C07285=1071.628,278.131,410.233,174.317,29.614,155.314
C07286=1071.623,277.882,410.263,174.314,29.610,155.313
C07287=1071.617,277.634,410.293,174.312,29.606,155.313
C07288=1071.611,277.386,410.322,174.309,29.602,155.312
C07289=1071.601,276.969,410.372,174.304,29.595,155.311
C07290=1071.591,276.552,410.422,174.300,29.588,155.310
C07291=1071.581,276.135,410.472,174.295,29.581,155.309
C07292=1071.570,275.717,410.522,174.291,29.575,155.307
C07293=1071.565,275.469,410.552,174.288,29.570,155.307
C07294=1071.558,275.221,410.581,174.285,29.567,155.306
C07295=1071.553,274.973,410.611,174.283,29.562,155.305
C07296=1071.547,274.725,410.640,174.280,29.558,155.305
C07297=1071.541,274.476,410.670,174.278,29.554,155.304
C07298=1071.535,274.228,410.699,174.275,29.550,155.303
C07299=1071.529,273.980,410.729,174.272,29.547,155.303
C07300=1071.523,273.732,410.758,174.270,29.542,155.302
C07301=1071.517,273.484,410.788,174.267,29.538,155.301
C07302=1071.512,273.236,410.817,174.264,29.534,155.301
C07303=1071.506,272.988,410.846,174.261,29.530,155.300
C07304=1071.500,272.740,410.875,174.259,29.526,155.299
C07305=1071.494,272.491,410.905,174.256,29.522,155.299
C07306=1071.488,272.243,410.934,174.254,29.518,155.298
C07307=1071.483,271.995,410.963,174.251,29.514,155.297
C07308=1071.476,271.747,410.992,174.249,29.510,155.297
C07309=1071.470,271.499,411.022,174.246,29.506,155.296
C07310=1071.465,271.250,411.051,174.244,29.502,155.295
C07311=1071.458,271.002,411.080,174.241,29.498,155.295
C07312=1071.452,270.754,411.109,174.239,29.494,155.294
C07313=1071.447,270.505,411.139,174.235,29.490,155.293
C07314=1071.440,270.257,411.168,174.233,29.486,155.293
C07315=1071.435,270.009,411.198,174.230,29.482,155.292
C07316=1071.429,269.761,411.227,174.228,29.478,155.291
C07317=1071.422,269.513,411.256,174.225,29.474,155.291
C07318=1071.417,269.264,411.285,174.223,29.470,155.290
C07319=1071.411,269.017,411.314,174.220,29.466,155.289
C07320=1071.405,268.769,411.343,174.218,29.462,155.289
C07321=1071.399,268.520,411.371,174.215,29.458,155.288
C07322=1071.393,268.271,411.401,174.213,29.455,155.287
C07323=1071.387,268.023,411.430,174.210,29.450,155.287
C07324=1071.381,267.775,411.459,174.208,29.446,155.286
C07325=1071.375,267.527,411.488,174.205,29.442,155.285
C07326=1071.369,267.278,411.516,174.202,29.438,155.285
C07327=1071.363,267.030,411.546,174.200,29.434,155.284
C07328=1071.358,266.782,411.575,174.197,29.431,155.283
C07329=1071.351,266.534,411.604,174.195,29.427,155.283
C07330=1071.345,266.286,411.632,174.191,29.422,155.282
C07331=1071.340,266.037,411.662,174.189,29.419,155.282
C07332=1071.334,265.789,411.691,174.186,29.415,155.281
C07333=1071.328,265.540,411.719,174.184,29.410,155.280
C07334=1071.322,265.293,411.748,174.181,29.406,155.279
C07335=1071.316,265.045,411.777,174.179,29.402,155.279
C07336=1071.310,264.796,411.805,174.176,29.398,155.278
C07337=1071.304,264.547,411.835,174.174,29.395,155.277
C07338=1071.299,264.300,411.863,174.171,29.391,155.277
C07339=1071.293,264.051,411.892,174.169,29.387,155.276
C07340=1071.287,263.803,411.921,174.166,29.383,155.276
C07341=1071.277,263.389,411.968,174.162,29.376,155.274
C07342=1071.266,262.976,412.016,174.158,29.370,155.273
C07343=1071.256,262.562,412.064,174.154,29.363,155.272
C07344=1071.246,262.148,412.111,174.150,29.357,155.271
C07345=1071.240,261.899,412.139,174.147,29.353,155.271
C07346=1071.234,261.651,412.168,174.145,29.349,155.270
C07347=1071.228,261.402,412.197,174.142,29.345,155.269
C07348=1071.222,261.155,412.225,174.140,29.341,155.269
C07349=1071.216,260.906,412.253,174.137,29.337,155.268
C07350=1071.209,260.658,412.282,174.134,29.333,155.267
C07351=1071.204,260.410,412.311,174.132,29.329,155.267
C07352=1071.198,260.162,412.339,174.129,29.325,155.266
C07353=1071.192,259.913,412.368,174.127,29.321,155.265
C07354=1071.186,259.665,412.396,174.124,29.317,155.265
C07355=1071.179,259.416,412.424,174.122,29.313,155.264
C07356=1071.174,259.169,412.452,174.119,29.310,155.264
C07357=1071.168,258.920,412.481,174.117,29.306,155.263
C07358=1071.162,258.671,412.509,174.114,29.302,155.262
C07359=1071.156,258.423,412.537,174.112,29.298,155.262
C07360=1071.150,258.175,412.566,174.109,29.294,155.261
C07361=1071.144,257.927,412.594,174.107,29.290,155.260
C07362=1071.138,257.678,412.622,174.104,29.286,155.260
C07363=1071.132,257.430,412.650,174.102,29.282,155.259
C07364=1071.126,257.182,412.679,174.099,29.278,155.258
C07365=1071.120,256.933,412.707,174.097,29.275,155.258
C07366=1071.114,256.685,412.735,174.094,29.271,155.257
C07367=1071.108,256.437,412.763,174.092,29.267,155.256
C07368=1071.102,256.188,412.791,174.089,29.263,155.256
C07369=1071.097,255.940,412.819,174.087,29.259,155.255
C07370=1071.091,255.691,412.848,174.084,29.255,155.254
C07371=1071.084,255.443,412.876,174.082,29.251,155.254
C07372=1071.078,255.195,412.904,174.079,29.246,155.253
C07373=1071.073,254.946,412.932,174.077,29.242,155.252
C07374=1071.067,254.698,412.960,174.074,29.239,155.252
C07375=1071.060,254.450,412.988,174.073,29.235,155.251
C07376=1071.055,254.201,413.016,174.070,29.231,155.250
C07377=1071.049,253.953,413.044,174.068,29.227,155.250
C07378=1071.043,253.704,413.073,174.065,29.223,155.249
C07379=1071.037,253.457,413.100,174.063,29.219,155.249
C07380=1071.031,253.208,413.128,174.060,29.215,155.248
C07381=1071.026,252.960,413.156,174.058,29.211,155.247
C07382=1071.020,252.711,413.185,174.055,29.207,155.247
C07383=1071.014,252.463,413.212,174.053,29.203,155.246
C07384=1071.008,252.214,413.240,174.050,29.199,155.245
C07385=1071.002,251.966,413.269,174.048,29.195,155.245
C07386=1070.997,251.718,413.297,174.045,29.191,155.244
C07387=1070.990,251.469,413.324,174.043,29.187,155.243
C07388=1070.985,251.221,413.352,174.041,29.183,155.243
C07389=1070.979,250.972,413.380,174.039,29.180,155.242
C07390=1070.973,250.724,413.407,174.036,29.176,155.241
C07391=1070.967,250.475,413.436,174.034,29.171,155.241
C07392=1070.962,250.227,413.464,174.032,29.167,155.240
C07393=1070.952,249.811,413.510,174.027,29.161,155.239
C07394=1070.943,249.395,413.556,174.023,29.154,155.238
C07395=1070.933,248.979,413.603,174.019,29.148,155.237
C07396=1070.923,248.562,413.649,174.015,29.140,155.236
C07397=1070.917,248.314,413.677,174.013,29.137,155.235
C07398=1070.911,248.066,413.705,174.011,29.133,155.234
C07399=1070.906,247.817,413.733,174.009,29.129,155.234
C07400=1070.900,247.569,413.760,174.006,29.125,155.233
C07401=1070.894,247.321,413.788,174.004,29.121,155.232
C07402=1070.888,247.072,413.816,174.001,29.117,155.232
C07403=1070.883,246.824,413.843,173.999,29.113,155.231
C07404=1070.877,246.575,413.871,173.996,29.109,155.230
C07405=1070.871,246.327,413.898,173.994,29.105,155.230
C07406=1070.865,246.078,413.926,173.991,29.101,155.229
C07407=1070.859,245.830,413.954,173.990,29.097,155.228
C07408=1070.853,245.582,413.980,173.987,29.093,155.228
C07409=1070.847,245.333,414.009,173.985,29.089,155.227
C07410=1070.841,245.085,414.035,173.982,29.085,155.226
C07411=1070.835,244.836,414.064,173.980,29.081,155.226
C07412=1070.830,244.587,414.090,173.977,29.077,155.225
C07413=1070.824,244.339,414.118,173.975,29.073,155.224
C07414=1070.818,244.090,414.145,173.973,29.069,155.224
C07415=1070.813,243.842,414.173,173.971,29.065,155.223
C07416=1070.807,243.594,414.200,173.968,29.061,155.222
C07417=1070.800,243.345,414.228,173.966,29.057,155.222
C07418=1070.795,243.097,414.255,173.964,29.053,155.221
C07419=1070.789,242.849,414.282,173.961,29.049,155.221
C07420=1070.783,242.600,414.310,173.959,29.046,155.220
C07421=1070.778,242.351,414.336,173.957,29.042,155.219
C07422=1070.771,242.103,414.364,173.955,29.038,155.219
C07423=1070.765,241.855,414.391,173.952,29.034,155.218
C07424=1070.760,241.606,414.419,173.950,29.030,155.217
C07425=1070.753,241.357,414.446,173.947,29.026,155.217
C07426=1070.748,241.109,414.472,173.945,29.022,155.216
C07427=1070.742,240.861,414.500,173.942,29.018,155.215
C07428=1070.735,240.612,414.527,173.941,29.014,155.215
C07429=1070.730,240.364,414.554,173.938,29.010,155.214
C07430=1070.724,240.115,414.581,173.936,29.006,155.213
C07431=1070.718,239.867,414.608,173.933,29.002,155.213
C07432=1070.712,239.618,414.635,173.931,28.998,155.212
C07433=1070.706,239.370,414.662,173.928,28.994,155.212
C07434=1070.701,239.121,414.689,173.927,28.991,155.211
C07435=1070.695,238.873,414.717,173.925,28.987,155.210
C07436=1070.689,238.625,414.743,173.922,28.983,155.210
C07437=1070.682,238.376,414.770,173.920,28.979,155.209
C07438=1070.677,238.127,414.797,173.917,28.975,155.208
C07439=1070.671,237.879,414.824,173.915,28.971,155.208
C07440=1070.665,237.631,414.851,173.913,28.967,155.207
C07441=1070.658,237.382,414.878,173.911,28.963,155.206
C07442=1070.653,237.133,414.905,173.908,28.959,155.206
C07443=1070.648,236.885,414.932,173.906,28.955,155.205
C07444=1070.642,236.637,414.959,173.903,28.951,155.204
C07445=1070.636,236.425,414.981,173.902,28.948,155.204
C07446=1070.631,236.214,415.005,173.900,28.945,155.203
C07447=1070.626,236.002,415.027,173.898,28.941,155.203
C07448=1070.621,235.791,415.050,173.896,28.938,155.202
C07449=1070.617,235.580,415.072,173.894,28.935,155.202
C07450=1070.612,235.368,415.095,173.892,28.931,155.201
C07451=1070.606,235.157,415.118,173.891,28.928,155.201
C07452=1070.601,234.945,415.141,173.888,28.924,155.200
C07453=1070.596,234.697,415.168,173.886,28.920,155.199
C07454=1070.590,234.449,415.195,173.884,28.916,155.199
C07455=1070.584,234.200,415.221,173.882,28.912,155.198
C07456=1070.578,233.952,415.248,173.879,28.908,155.197
C07457=1070.573,233.704,415.275,173.877,28.905,155.197
C07458=1070.566,233.454,415.302,173.875,28.901,155.196
C07459=1070.560,233.206,415.328,173.873,28.897,155.195
C07460=1070.555,232.958,415.355,173.870,28.893,155.195
C07461=1070.549,232.709,415.381,173.868,28.889,155.194
C07462=1070.543,232.460,415.408,173.865,28.885,155.194
C07463=1070.537,232.211,415.435,173.864,28.881,155.193
C07464=1070.531,231.963,415.461,173.861,28.877,155.192
C07465=1070.525,231.715,415.488,173.859,28.873,155.192
C07466=1070.520,231.466,415.515,173.857,28.869,155.191
C07467=1070.514,231.218,415.541,173.855,28.865,155.190
C07468=1070.508,230.969,415.567,173.853,28.861,155.190
C07469=1070.503,230.721,415.594,173.850,28.857,155.189
C07470=1070.497,230.472,415.620,173.848,28.853,155.188
C07471=1070.491,230.223,415.647,173.845,28.849,155.188
C07472=1070.484,229.975,415.673,173.844,28.845,155.187
C07473=1070.479,229.726,415.699,173.841,28.841,155.186
C07474=1070.473,229.478,415.726,173.839,28.837,155.186
C07475=1070.467,229.229,415.753,173.837,28.833,155.185
C07476=1070.462,228.980,415.779,173.835,28.829,155.184
C07477=1070.455,228.732,415.805,173.833,28.825,155.184
C07478=1070.449,228.483,415.832,173.830,28.821,155.183
C07479=1070.443,228.234,415.858,173.828,28.817,155.182
C07480=1070.437,227.986,415.884,173.826,28.814,155.182
C07481=1070.431,227.738,415.910,173.824,28.810,155.181
C07482=1070.425,227.489,415.936,173.821,28.806,155.180
C07483=1070.420,227.241,415.963,173.819,28.802,155.180
C07484=1070.413,226.993,415.989,173.818,28.798,155.179
C07485=1070.408,226.744,416.015,173.815,28.794,155.179
C07486=1070.402,226.495,416.042,173.813,28.790,155.178
C07487=1070.396,226.246,416.067,173.810,28.786,155.177
C07488=1070.390,225.998,416.094,173.809,28.782,155.177
C07489=1070.384,225.749,416.119,173.806,28.778,155.176
C07490=1070.379,225.501,416.146,173.804,28.774,155.175
C07491=1070.372,225.252,416.171,173.802,28.770,155.175
C07492=1070.367,225.004,416.198,173.800,28.766,155.174
C07493=1070.361,224.755,416.224,173.798,28.762,155.173
C07494=1070.355,224.507,416.250,173.795,28.758,155.173
C07495=1070.349,224.258,416.276,173.794,28.755,155.172
C07496=1070.343,224.009,416.303,173.791,28.750,155.171
C07497=1070.337,223.761,416.328,173.789,28.746,155.171
C07498=1070.332,223.512,416.355,173.787,28.743,155.170
C07499=1070.326,223.263,416.381,173.785,28.739,155.170
C07500=1070.320,223.015,416.407,173.782,28.735,155.169
C07501=1070.315,222.799,416.429,173.781,28.731,155.168
C07502=1070.310,222.585,416.452,173.779,28.727,155.168
C07503=1070.305,222.368,416.474,173.777,28.724,155.167
C07504=1070.299,222.153,416.497,173.775,28.720,155.166
C07505=1070.295,221.938,416.519,173.773,28.717,155.166
C07506=1070.290,221.722,416.542,173.771,28.714,155.165
C07507=1070.285,221.507,416.564,173.770,28.711,155.165
C07508=1070.280,221.291,416.587,173.767,28.707,155.164
C07509=1070.273,221.043,416.613,173.766,28.703,155.164
C07510=1070.268,220.794,416.638,173.764,28.699,155.163
C07511=1070.262,220.545,416.664,173.761,28.695,155.162
C07512=1070.256,220.296,416.690,173.760,28.691,155.162
C07513=1070.250,220.048,416.716,173.757,28.687,155.161
C07514=1070.243,219.800,416.741,173.755,28.683,155.160
C07515=1070.238,219.551,416.767,173.753,28.679,155.160
C07516=1070.232,219.302,416.792,173.751,28.675,155.159
C07517=1070.226,219.054,416.819,173.749,28.671,155.158
C07518=1070.220,218.805,416.844,173.746,28.667,155.158
C07519=1070.214,218.556,416.870,173.745,28.663,155.157
C07520=1070.209,218.308,416.895,173.742,28.659,155.157
C07521=1070.202,218.059,416.921,173.740,28.655,155.156
C07522=1070.197,217.810,416.947,173.738,28.652,155.155
C07523=1070.190,217.562,416.973,173.736,28.648,155.155
C07524=1070.185,217.313,416.999,173.734,28.644,155.154
C07525=1070.179,217.065,417.024,173.732,28.640,155.153
C07526=1070.173,216.816,417.049,173.730,28.636,155.153
C07527=1070.167,216.567,417.075,173.727,28.631,155.152
C07528=1070.162,216.319,417.100,173.726,28.627,155.151
C07529=1070.156,216.070,417.126,173.724,28.623,155.151
C07530=1070.150,215.822,417.151,173.721,28.619,155.150
C07531=1070.144,215.573,417.177,173.720,28.616,155.149
C07532=1070.138,215.324,417.203,173.717,28.612,155.149
C07533=1070.132,215.075,417.228,173.715,28.608,155.148
C07534=1070.126,214.827,417.253,173.713,28.604,155.147
C07535=1070.121,214.578,417.279,173.711,28.600,155.147
C07536=1070.115,214.330,417.304,173.709,28.595,155.146
C07537=1070.108,214.081,417.330,173.707,28.591,155.145
C07538=1070.103,213.832,417.356,173.705,28.587,155.145
C07539=1070.097,213.584,417.381,173.703,28.584,155.144
C07540=1070.092,213.335,417.406,173.701,28.580,155.143
C07541=1070.086,213.086,417.432,173.699,28.576,155.143
C07542=1070.080,212.838,417.457,173.697,28.571,155.142
C07543=1070.074,212.590,417.482,173.695,28.567,155.141
C07544=1070.068,212.341,417.508,173.692,28.563,155.141
C07545=1070.062,212.092,417.533,173.691,28.559,155.140
C07546=1070.056,211.843,417.558,173.688,28.555,155.139
C07547=1070.050,211.594,417.583,173.686,28.551,155.139
C07548=1070.045,211.346,417.608,173.685,28.547,155.138
C07549=1070.039,211.097,417.634,173.682,28.543,155.137
C07550=1070.033,210.848,417.660,173.681,28.540,155.137
C07551=1070.027,210.600,417.685,173.678,28.535,155.136
C07552=1070.021,210.351,417.709,173.676,28.531,155.135
C07553=1070.015,210.103,417.734,173.675,28.527,155.135
C07554=1070.009,209.854,417.760,173.672,28.523,155.134
C07555=1070.003,209.605,417.785,173.670,28.519,155.133
C07556=1069.998,209.356,417.810,173.668,28.515,155.133
C07557=1069.992,209.144,417.832,173.667,28.512,155.132
C07558=1069.987,208.930,417.853,173.664,28.508,155.132
C07559=1069.983,208.717,417.875,173.663,28.505,155.131
C07560=1069.977,208.504,417.896,173.661,28.502,155.131
C07561=1069.972,208.291,417.917,173.660,28.498,155.130
C07562=1069.968,208.077,417.939,173.658,28.494,155.129
C07563=1069.962,207.864,417.960,173.656,28.491,155.129
C07564=1069.957,207.652,417.982,173.654,28.488,155.128
C07565=1069.933,206.608,418.085,173.515,28.417,155.126
C07566=1069.928,206.359,418.109,173.513,28.413,155.125
C07567=1069.922,206.111,418.133,173.511,28.410,155.125
C07568=1069.916,205.862,418.157,173.509,28.407,155.124
C07569=1069.910,205.613,418.182,173.506,28.404,155.124
C07570=1069.905,205.364,418.206,173.504,28.401,155.123
C07571=1069.898,205.116,418.230,173.502,28.398,155.123
C07572=1069.893,204.867,418.254,173.500,28.395,155.122
C07573=1069.887,204.618,418.279,173.497,28.392,155.122
C07574=1069.882,204.369,418.303,173.496,28.389,155.121
C07575=1069.876,204.121,418.327,173.493,28.386,155.121
C07576=1069.870,203.872,418.351,173.491,28.382,155.121
C07577=1069.865,203.623,418.375,173.489,28.379,155.120
C07578=1069.859,203.374,418.400,173.487,28.377,155.120
C07579=1069.853,203.126,418.423,173.484,28.373,155.119
C07580=1069.848,202.876,418.447,173.482,28.370,155.119
C07581=1069.843,202.628,418.472,173.480,28.367,155.118
C07582=1069.837,202.379,418.496,173.477,28.364,155.118
C07583=1069.831,202.130,418.520,173.476,28.361,155.118
C07584=1069.825,201.881,418.544,173.473,28.358,155.117
C07585=1069.819,201.633,418.568,173.471,28.355,155.117
C07586=1069.813,201.384,418.592,173.469,28.352,155.116
C07587=1069.808,201.135,418.615,173.467,28.349,155.116
C07588=1069.802,200.886,418.640,173.464,28.346,155.115
C07589=1069.796,200.637,418.664,173.463,28.343,155.115
C07590=1069.790,200.389,418.688,173.460,28.340,155.115
C07591=1069.784,200.141,418.712,173.458,28.337,155.114
C07592=1069.778,199.891,418.735,173.456,28.334,155.114
C07593=1069.773,199.642,418.759,173.454,28.331,155.113
C07594=1069.767,199.394,418.783,173.451,28.328,155.113
C07595=1069.761,199.145,418.807,173.450,28.325,155.112
C07596=1069.755,198.896,418.830,173.447,28.322,155.112
C07597=1069.750,198.647,418.855,173.444,28.319,155.112
C07598=1069.743,198.398,418.879,173.443,28.316,155.111
C07599=1069.738,198.149,418.902,173.440,28.313,155.111
C07600=1069.732,197.901,418.926,173.439,28.310,155.110
C07601=1069.727,197.652,418.950,173.436,28.307,155.110
C07602=1069.720,197.403,418.973,173.434,28.304,155.109
C07603=1069.714,197.154,418.997,173.432,28.301,155.109
C07604=1069.709,196.906,419.021,173.430,28.298,155.109
C07605=1069.703,196.657,419.044,173.427,28.295,155.108
C07606=1069.697,196.408,419.069,173.426,28.292,155.108
C07607=1069.691,196.159,419.093,173.423,28.289,155.107
C07608=1069.686,195.910,419.115,173.422,28.286,155.107
C07609=1069.680,195.662,419.140,173.419,28.283,155.107
C07610=1069.675,195.413,419.163,173.417,28.280,155.106
C07611=1069.669,195.164,419.187,173.415,28.277,155.106
C07612=1069.663,194.915,419.210,173.413,28.274,155.105
C07613=1069.658,194.666,419.235,173.411,28.271,155.105
C07614=1069.652,194.417,419.257,173.408,28.268,155.104
C07615=1069.646,194.169,419.281,173.406,28.265,155.104
C07616=1069.641,193.920,419.305,173.404,28.262,155.103
C07617=1069.634,193.671,419.329,173.402,28.259,155.103
C07618=1069.629,193.422,419.352,173.400,28.256,155.103
C07619=1069.623,193.173,419.376,173.398,28.253,155.102
C07620=1069.618,192.924,419.399,173.395,28.250,155.102
C07621=1069.612,192.676,419.423,173.394,28.247,155.101
C07622=1069.607,192.427,419.446,173.391,28.244,155.101
C07623=1069.601,192.179,419.470,173.390,28.241,155.101
C07624=1069.595,191.929,419.494,173.387,28.238,155.100
C07625=1069.589,191.681,419.517,173.386,28.235,155.100
C07626=1069.583,191.399,419.544,173.383,28.232,155.099
C07627=1069.576,191.117,419.570,173.381,28.229,155.099
C07628=1069.569,190.834,419.597,173.378,28.225,155.098
C07629=1069.564,190.552,419.624,173.376,28.222,155.098
C07630=1069.558,190.303,419.647,173.373,28.219,155.097
C07631=1069.552,190.055,419.670,173.372,28.216,155.097
C07632=1069.547,189.806,419.694,173.369,28.213,155.097
C07633=1069.541,189.557,419.717,173.368,28.210,155.096
C07634=1069.536,189.308,419.740,173.365,28.207,155.096
C07635=1069.531,189.059,419.763,173.364,28.204,155.095
C07636=1069.525,188.811,419.787,173.361,28.201,155.095
C07637=1069.519,188.562,419.810,173.359,28.197,155.094
C07638=1069.514,188.313,419.833,173.357,28.195,155.094
C07639=1069.508,188.064,419.857,173.355,28.192,155.094
C07640=1069.502,187.815,419.880,173.353,28.189,155.093
C07641=1069.496,187.567,419.903,173.351,28.186,155.093
C07642=1069.491,187.317,419.927,173.349,28.183,155.092
C07643=1069.486,187.068,419.950,173.347,28.180,155.092
C07644=1069.480,186.820,419.973,173.345,28.177,155.091
C07645=1069.475,186.571,419.997,173.342,28.174,155.091
C07646=1069.469,186.322,420.020,173.341,28.171,155.091
C07647=1069.463,186.073,420.043,173.338,28.168,155.090
C07648=1069.457,185.824,420.066,173.337,28.165,155.090
C07649=1069.452,185.576,420.090,173.334,28.162,155.089
C07650=1069.446,185.327,420.113,173.333,28.159,155.089
C07651=1069.441,185.078,420.136,173.330,28.156,155.088
C07652=1069.436,184.829,420.159,173.329,28.153,155.088
C07653=1069.430,184.580,420.182,173.326,28.150,155.088
C07654=1069.423,184.331,420.205,173.325,28.147,155.087
C07655=1069.418,184.082,420.227,173.322,28.144,155.087
C07656=1069.412,183.833,420.250,173.321,28.142,155.086
C07657=1069.406,183.584,420.274,173.318,28.139,155.086
C07658=1069.400,183.335,420.297,173.316,28.136,155.086
C07659=1069.394,183.086,420.320,173.314,28.133,155.085
C07660=1069.388,182.837,420.343,173.312,28.130,155.085
C07661=1069.382,182.589,420.365,173.310,28.127,155.084
C07662=1069.376,182.340,420.388,173.307,28.124,155.084
C07663=1069.371,182.091,420.411,173.306,28.122,155.084
C07664=1069.365,181.842,420.434,173.303,28.119,155.083
C07665=1069.359,181.593,420.457,173.302,28.116,155.083
C07666=1069.353,181.344,420.480,173.299,28.113,155.082
C07667=1069.347,181.095,420.502,173.298,28.110,155.082
C07668=1069.341,180.847,420.525,173.295,28.108,155.082
C07669=1069.335,180.598,420.548,173.294,28.105,155.081
C07670=1069.330,180.349,420.571,173.291,28.102,155.081
C07671=1069.324,180.099,420.593,173.290,28.099,155.081
C07672=1069.318,179.851,420.615,173.288,28.097,155.080
C07673=1069.312,179.602,420.638,173.285,28.094,155.080
C07674=1069.306,179.353,420.661,173.284,28.091,155.079
C07675=1069.301,179.104,420.684,173.281,28.088,155.079
C07676=1069.295,178.855,420.707,173.280,28.085,155.079
C07677=1069.288,178.606,420.730,173.277,28.082,155.078
C07678=1069.283,178.357,420.752,173.276,28.079,155.078
C07679=1069.278,178.109,420.774,173.273,28.076,155.077
C07680=1069.272,177.860,420.797,173.272,28.074,155.077
C07681=1069.266,177.611,420.820,173.269,28.071,155.077
C07682=1069.260,177.362,420.843,173.268,28.068,155.076
C07683=1069.255,177.113,420.865,173.265,28.065,155.076
C07684=1069.249,176.864,420.888,173.264,28.062,155.075
C07685=1069.243,176.615,420.911,173.261,28.059,155.075
C07686=1069.237,176.367,420.933,173.260,28.057,155.075
C07687=1069.231,176.117,420.955,173.258,28.054,155.074
C07688=1069.225,175.868,420.978,173.255,28.051,155.074
C07689=1069.220,175.620,421.001,173.254,28.048,155.073
C07690=1069.212,175.277,421.031,173.251,28.044,155.073
C07691=1069.204,174.935,421.062,173.248,28.040,155.072
C07692=1069.196,174.592,421.094,173.246,28.036,155.072
C07693=1069.188,174.251,421.124,173.243,28.032,155.071
C07694=1069.183,174.001,421.146,173.241,28.030,155.071
C07695=1069.177,173.752,421.169,173.238,28.027,155.070
C07696=1069.171,173.503,421.192,173.237,28.024,155.070
C07697=1069.165,173.254,421.214,173.234,28.021,155.070
C07698=1069.160,173.006,421.237,173.233,28.018,155.069
C07699=1069.155,172.756,421.259,173.231,28.015,155.069
C07700=1069.148,172.508,421.281,173.229,28.012,155.068
C07701=1069.142,172.259,421.304,173.227,28.010,155.068
C07702=1069.137,172.009,421.326,173.225,28.007,155.068
C07703=1069.131,171.762,421.348,173.223,28.004,155.067
C07704=1069.126,171.512,421.371,173.222,28.001,155.067
C07705=1069.120,171.263,421.393,173.219,27.998,155.066
C07706=1069.115,171.014,421.416,173.218,27.995,155.066
C07707=1069.108,170.765,421.438,173.215,27.992,155.066
C07708=1069.103,170.516,421.460,173.214,27.990,155.065
C07709=1069.098,170.267,421.483,173.212,27.987,155.065
C07710=1069.091,170.018,421.505,173.210,27.984,155.064
C07711=1069.086,169.770,421.527,173.208,27.981,155.064
C07712=1069.081,169.520,421.549,173.205,27.978,155.064
C07713=1069.074,169.272,421.572,173.204,27.975,155.063
C07714=1069.069,169.022,421.594,173.202,27.972,155.063
C07715=1069.064,168.774,421.616,173.200,27.969,155.062
C07716=1069.058,168.525,421.638,173.198,27.966,155.062
C07717=1069.052,168.275,421.660,173.196,27.963,155.062
C07718=1069.047,168.056,421.680,173.194,27.961,155.061
C07719=1069.042,167.838,421.700,173.193,27.958,155.061
C07720=1069.037,167.619,421.719,173.191,27.956,155.061
C07721=1069.032,167.400,421.739,173.190,27.954,155.060
C07722=1069.028,167.181,421.759,173.188,27.951,155.060
C07723=1069.023,166.962,421.778,173.186,27.949,155.059
C07724=1069.018,166.743,421.798,173.185,27.946,155.059
C07725=1069.013,166.524,421.817,173.183,27.944,155.059
C07726=1069.008,166.275,421.839,173.181,27.941,155.058
C07727=1069.002,166.026,421.860,173.179,27.938,155.058
C07728=1068.996,165.777,421.883,173.178,27.935,155.058
C07729=1068.990,165.528,421.905,173.175,27.932,155.057
C07730=1068.985,165.279,421.927,173.174,27.929,155.057
C07731=1068.979,165.030,421.950,173.171,27.926,155.056
C07732=1068.974,164.781,421.971,173.170,27.923,155.056
C07733=1068.968,164.532,421.993,173.168,27.920,155.055
C07734=1068.963,164.283,422.015,173.166,27.917,155.055
C07735=1068.957,164.034,422.038,173.164,27.915,155.055
C07736=1068.951,163.785,422.060,173.162,27.912,155.054
C07737=1068.946,163.536,422.081,173.160,27.909,155.054
C07738=1068.940,163.287,422.103,173.158,27.906,155.053
C07739=1068.935,163.038,422.125,173.157,27.903,155.053
C07740=1068.929,162.789,422.148,173.154,27.900,155.053
C07741=1068.924,162.540,422.170,173.153,27.898,155.052
C07742=1068.918,162.291,422.191,173.151,27.895,155.052
C07743=1068.913,162.042,422.213,173.149,27.892,155.051
C07744=1068.907,161.793,422.235,173.147,27.889,155.051
C07745=1068.901,161.544,422.257,173.146,27.886,155.051
C07746=1068.897,161.296,422.279,173.143,27.883,155.050
C07747=1068.890,161.046,422.301,173.142,27.880,155.050
C07748=1068.884,160.797,422.323,173.140,27.878,155.049
C07749=1068.879,160.549,422.344,173.138,27.875,155.049
C07750=1068.873,160.299,422.366,173.136,27.872,155.049
C07751=1068.867,160.050,422.388,173.135,27.869,155.048
C07752=1068.862,159.802,422.409,173.132,27.866,155.048
C07753=1068.856,159.552,422.431,173.131,27.864,155.047
C07754=1068.850,159.269,422.456,173.128,27.861,155.047
C07755=1068.843,158.987,422.480,173.127,27.857,155.047
C07756=1068.836,158.704,422.505,173.124,27.854,155.046
C07757=1068.830,158.421,422.530,173.122,27.851,155.046
C07758=1068.824,158.173,422.551,173.120,27.848,155.045
C07759=1068.818,157.923,422.573,173.119,27.845,155.045
C07760=1068.813,157.675,422.594,173.116,27.842,155.044
C07761=1068.807,157.425,422.616,173.115,27.840,155.044
C07762=1068.801,157.176,422.638,173.113,27.837,155.044
C07763=1068.795,156.928,422.659,173.112,27.834,155.043
C07764=1068.790,156.677,422.681,173.109,27.831,155.043
C07765=1068.784,156.429,422.702,173.108,27.829,155.043
C07766=1068.778,156.180,422.723,173.106,27.826,155.042
C07767=1068.773,155.931,422.745,173.104,27.823,155.042
C07768=1068.767,155.682,422.767,173.102,27.820,155.041
C07769=1068.762,155.433,422.788,173.100,27.817,155.041
C07770=1068.756,155.184,422.810,173.098,27.814,155.041
C07771=1068.750,154.936,422.831,173.096,27.812,155.040
C07772=1068.744,154.686,422.853,173.095,27.809,155.040
C07773=1068.738,154.437,422.874,173.093,27.807,155.040
C07774=1068.732,154.188,422.895,173.091,27.804,155.039
C07775=1068.726,153.939,422.917,173.089,27.801,155.039
C07776=1068.721,153.690,422.938,173.088,27.798,155.038
C07777=1068.715,153.441,422.960,173.085,27.795,155.038
C07778=1068.710,153.192,422.981,173.084,27.792,155.038
C07779=1068.704,152.942,423.002,173.082,27.790,155.037
C07780=1068.698,152.694,423.024,173.081,27.787,155.037
C07781=1068.692,152.445,423.045,173.078,27.784,155.036
C07782=1068.687,152.196,423.066,173.077,27.781,155.036
C07783=1068.681,151.946,423.087,173.075,27.779,155.036
C07784=1068.675,151.698,423.109,173.073,27.776,155.035
C07785=1068.669,151.449,423.130,173.071,27.773,155.035
C07786=1068.663,151.200,423.152,173.069,27.770,155.034
C07787=1068.658,150.950,423.173,173.068,27.768,155.034
C07788=1068.653,150.702,423.194,173.065,27.765,155.034
C07789=1068.647,150.453,423.216,173.064,27.762,155.033
C07790=1068.641,150.203,423.237,173.062,27.759,155.033
C07791=1068.636,149.955,423.258,173.060,27.756,155.032
C07792=1068.630,149.706,423.279,173.058,27.753,155.032
C07793=1068.624,149.456,423.300,173.057,27.750,155.032
C07794=1068.618,149.207,423.322,173.055,27.748,155.031
C07795=1068.613,148.959,423.343,173.053,27.745,155.031
C07796=1068.607,148.709,423.364,173.051,27.742,155.031
C07797=1068.601,148.460,423.385,173.050,27.740,155.030
C07798=1068.596,148.211,423.406,173.048,27.737,155.030
C07799=1068.590,147.962,423.427,173.046,27.734,155.029
C07800=1068.583,147.714,423.448,173.044,27.731,155.029
C07801=1068.578,147.464,423.469,173.043,27.728,155.029
C07802=1068.572,147.216,423.490,173.041,27.726,155.028
C07803=1068.566,146.966,423.511,173.039,27.723,155.028
C07804=1068.561,146.717,423.532,173.037,27.720,155.027
C07805=1068.555,146.467,423.553,173.036,27.718,155.027
C07806=1068.549,146.219,423.574,173.034,27.715,155.027
C07807=1068.543,145.970,423.594,173.032,27.712,155.026
C07808=1068.537,145.721,423.616,173.030,27.709,155.026
C07809=1068.532,145.472,423.637,173.029,27.706,155.025
C07810=1068.526,145.223,423.658,173.027,27.704,155.025
C07811=1068.520,144.973,423.679,173.024,27.701,155.025
C07812=1068.515,144.725,423.700,173.023,27.698,155.024
C07813=1068.508,144.475,423.720,173.021,27.696,155.024
C07814=1068.503,144.227,423.742,173.020,27.693,155.024
C07815=1068.497,143.977,423.763,173.018,27.690,155.023
C07816=1068.491,143.729,423.784,173.016,27.687,155.023
C07817=1068.486,143.479,423.804,173.014,27.685,155.023
C07818=1068.479,143.196,423.827,173.013,27.681,155.022
C07819=1068.473,142.914,423.852,173.010,27.678,155.022
C07820=1068.466,142.630,423.876,173.008,27.675,155.021
C07821=1068.459,142.347,423.899,173.006,27.672,155.021
C07822=1068.454,142.098,423.920,173.005,27.669,155.020
C07823=1068.448,141.849,423.941,173.003,27.666,155.020
C07824=1068.442,141.599,423.962,173.001,27.663,155.020
C07825=1068.437,141.351,423.983,172.999,27.661,155.019
C07826=1068.431,141.102,424.003,172.998,27.658,155.019
C07827=1068.425,140.852,424.024,172.996,27.655,155.018
C07828=1068.420,140.603,424.045,172.994,27.653,155.018
C07829=1068.414,140.354,424.066,172.992,27.650,155.018
C07830=1068.408,140.106,424.086,172.991,27.647,155.017
C07831=1068.402,139.856,424.107,172.989,27.644,155.017
C07832=1068.397,139.607,424.128,172.988,27.642,155.016
C07833=1068.391,139.358,424.148,172.985,27.639,155.016
C07834=1068.385,139.109,424.169,172.984,27.636,155.016
C07835=1068.379,138.860,424.190,172.982,27.634,155.015
C07836=1068.373,138.611,424.210,172.981,27.631,155.015
C07837=1068.368,138.361,424.231,172.979,27.628,155.015
C07838=1068.362,138.112,424.251,172.977,27.625,155.014
C07839=1068.356,137.864,424.272,172.975,27.622,155.014
C07840=1068.350,137.614,424.293,172.974,27.619,155.013
C07841=1068.345,137.365,424.313,172.972,27.617,155.013
C07842=1068.339,137.116,424.333,172.971,27.614,155.013
C07843=1068.334,136.867,424.354,172.968,27.611,155.012
C07844=1068.327,136.618,424.374,172.967,27.609,155.012
C07845=1068.322,136.369,424.396,172.965,27.606,155.011
C07846=1068.316,136.120,424.416,172.964,27.603,155.011
C07847=1068.310,135.871,424.436,172.962,27.600,155.011
C07848=1068.304,135.621,424.457,172.960,27.598,155.010
C07849=1068.298,135.373,424.477,172.958,27.595,155.010
C07850=1068.293,135.124,424.498,172.956,27.592,155.010
C07851=1068.287,134.875,424.517,172.955,27.590,155.009
C07852=1068.281,134.625,424.538,172.953,27.587,155.009
C07853=1068.275,134.377,424.559,172.952,27.584,155.008
C07854=1068.270,134.128,424.580,172.949,27.581,155.008
C07855=1068.264,133.879,424.600,172.948,27.578,155.008
C07856=1068.258,133.629,424.620,172.946,27.576,155.007
C07857=1068.253,133.380,424.641,172.945,27.573,155.007
C07858=1068.247,133.131,424.661,172.943,27.570,155.007
C07859=1068.241,132.882,424.682,172.942,27.568,155.006
C07860=1068.235,132.633,424.702,172.939,27.565,155.006
C07861=1068.230,132.383,424.722,172.938,27.562,155.005
C07862=1068.224,132.134,424.742,172.936,27.559,155.005
C07863=1068.218,131.885,424.763,172.935,27.556,155.005
C07864=1068.212,131.636,424.783,172.933,27.554,155.004
C07865=1068.206,131.387,424.803,172.932,27.551,155.004
C07866=1068.200,131.138,424.824,172.929,27.548,155.003
C07867=1068.194,130.889,424.844,172.928,27.545,155.003
C07868=1068.188,130.640,424.864,172.926,27.543,155.003
C07869=1068.183,130.391,424.883,172.925,27.540,155.002
C07870=1068.177,130.141,424.904,172.923,27.538,155.002
C07871=1068.171,129.892,424.924,172.922,27.535,155.002
C07872=1068.165,129.643,424.944,172.919,27.532,155.001
C07873=1068.160,129.394,424.964,172.918,27.530,155.001
C07874=1068.153,129.145,424.985,172.916,27.527,155.000
C07875=1068.147,128.896,425.005,172.915,27.524,155.000
C07876=1068.141,128.647,425.025,172.913,27.521,155.000
C07877=1068.136,128.398,425.045,172.911,27.519,154.999
C07878=1068.130,128.149,425.064,172.910,27.516,154.999
C07879=1068.124,127.899,425.085,172.907,27.513,154.999
C07880=1068.118,127.650,425.105,172.906,27.510,154.998
C07881=1068.112,127.401,425.125,172.904,27.508,154.998
C07882=1068.106,127.117,425.148,172.903,27.505,154.997
C07883=1068.099,126.834,425.171,172.900,27.502,154.997
C07884=1068.092,126.551,425.194,172.899,27.498,154.996
C07885=1068.086,126.268,425.216,172.897,27.495,154.996
C07886=1068.079,126.019,425.236,172.895,27.493,154.996
C07887=1068.073,125.770,425.256,172.894,27.490,154.995
C07888=1068.068,125.521,425.276,172.892,27.488,154.995
C07889=1068.063,125.272,425.296,172.891,27.485,154.995
C07890=1068.057,125.023,425.316,172.889,27.482,154.994
C07891=1068.051,124.774,425.336,172.888,27.479,154.994
C07892=1068.046,124.524,425.355,172.885,27.476,154.993
C07893=1068.040,124.275,425.375,172.884,27.473,154.993
C07894=1068.033,124.026,425.396,172.882,27.471,154.993
C07895=1068.027,123.777,425.416,172.880,27.468,154.992
C07896=1068.021,123.528,425.435,172.879,27.466,154.992
C07897=1068.016,123.278,425.455,172.877,27.463,154.992
C07898=1068.010,123.030,425.475,172.876,27.460,154.991
C07899=1068.004,122.780,425.495,172.874,27.457,154.991
C07900=1067.998,122.531,425.515,172.872,27.454,154.990
C07901=1067.993,122.282,425.534,172.870,27.452,154.990
C07902=1067.987,122.033,425.554,172.869,27.449,154.990
C07903=1067.981,121.784,425.574,172.867,27.446,154.989
C07904=1067.976,121.535,425.594,172.866,27.444,154.989
C07905=1067.970,121.286,425.614,172.864,27.441,154.988
C07906=1067.964,121.037,425.634,172.863,27.438,154.988
C07907=1067.959,120.787,425.653,172.861,27.435,154.988
C07908=1067.953,120.538,425.673,172.859,27.432,154.987
C07909=1067.947,120.289,425.693,172.857,27.430,154.987
C07910=1067.941,120.040,425.713,172.856,27.427,154.987
C07911=1067.935,119.791,425.732,172.854,27.424,154.986
C07912=1067.930,119.542,425.752,172.853,27.422,154.986
C07913=1067.925,119.292,425.772,172.851,27.419,154.985
C07914=1067.919,119.043,425.792,172.850,27.416,154.985
C07915=1067.913,118.795,425.812,172.848,27.413,154.985
C07916=1067.907,118.545,425.831,172.847,27.410,154.984
C07917=1067.901,118.296,425.851,172.845,27.408,154.984
C07918=1067.895,118.047,425.870,172.843,27.405,154.983
C07919=1067.890,117.797,425.890,172.841,27.402,154.983
C07920=1067.884,117.548,425.910,172.840,27.400,154.983
C07921=1067.879,117.299,425.929,172.838,27.397,154.982
C07922=1067.873,117.050,425.949,172.837,27.394,154.982
C07923=1067.867,116.801,425.968,172.835,27.391,154.981
C07924=1067.861,116.552,425.988,172.834,27.388,154.981
C07925=1067.855,116.302,426.007,172.832,27.386,154.981
C07926=1067.850,116.053,426.028,172.831,27.383,154.980
C07927=1067.844,115.804,426.047,172.829,27.380,154.980
C07928=1067.839,115.554,426.066,172.828,27.377,154.979
C07929=1067.833,115.306,426.086,172.825,27.374,154.979
C07930=1067.827,115.056,426.106,172.824,27.371,154.979
C07931=1067.821,114.807,426.126,172.822,27.369,154.978
C07932=1067.816,114.559,426.144,172.821,27.366,154.978
C07933=1067.810,114.309,426.164,172.819,27.363,154.977
C07934=1067.804,114.060,426.184,172.818,27.361,154.977
C07935=1067.798,113.811,426.203,172.816,27.358,154.977
C07936=1067.793,113.562,426.222,172.815,27.355,154.976
C07937=1067.787,113.313,426.242,172.813,27.352,154.976
C07938=1067.781,113.063,426.261,172.812,27.350,154.976
C07939=1067.775,112.814,426.281,172.810,27.347,154.975
C07940=1067.769,112.565,426.301,172.809,27.345,154.975
C07941=1067.764,112.316,426.320,172.806,27.341,154.975
C07942=1067.758,112.066,426.339,172.805,27.339,154.974
C07943=1067.752,111.817,426.358,172.803,27.336,154.974
C07944=1067.746,111.568,426.378,172.802,27.333,154.973
C07945=1067.740,111.319,426.397,172.800,27.330,154.973
C07946=1067.734,111.036,426.419,172.799,27.328,154.972
C07947=1067.727,110.753,426.441,172.797,27.324,154.972
C07948=1067.720,110.469,426.463,172.795,27.321,154.972
C07949=1067.713,110.186,426.484,172.794,27.318,154.971
C07950=1067.708,109.937,426.504,172.792,27.315,154.971
C07951=1067.702,109.687,426.523,172.791,27.313,154.970
C07952=1067.696,109.438,426.542,172.789,27.310,154.970
C07953=1067.690,109.189,426.561,172.787,27.307,154.970
C07954=1067.684,108.939,426.580,172.785,27.305,154.969
C07955=1067.678,108.691,426.600,172.784,27.302,154.969
C07956=1067.673,108.441,426.619,172.782,27.299,154.969
C07957=1067.667,108.192,426.638,172.781,27.297,154.968
C07958=1067.661,107.943,426.657,172.779,27.294,154.968
C07959=1067.655,107.694,426.676,172.778,27.291,154.967
C07960=1067.650,107.444,426.695,172.776,27.288,154.967
C07961=1067.643,107.195,426.714,172.775,27.286,154.967
C07962=1067.638,106.946,426.733,172.773,27.283,154.966
C07963=1067.632,106.696,426.752,172.772,27.281,154.966
C07964=1067.626,106.448,426.772,172.770,27.278,154.966
C07965=1067.619,106.198,426.791,172.769,27.275,154.965
C07966=1067.614,105.950,426.810,172.767,27.272,154.965
C07967=1067.609,105.700,426.829,172.766,27.269,154.964
C07968=1067.603,105.451,426.848,172.764,27.266,154.964
C07969=1067.597,105.202,426.867,172.762,27.263,154.964
C07970=1067.591,104.952,426.886,172.760,27.261,154.963
C07971=1067.585,104.703,426.905,172.759,27.258,154.963
C07972=1067.579,104.454,426.924,172.757,27.256,154.962
C07973=1067.574,104.205,426.943,172.756,27.253,154.962
C07974=1067.568,103.956,426.962,172.754,27.250,154.962
C07975=1067.562,103.706,426.981,172.753,27.247,154.961
C07976=1067.556,103.457,427.000,172.751,27.244,154.961
C07977=1067.551,103.208,427.019,172.750,27.242,154.960
C07978=1067.545,102.959,427.038,172.748,27.239,154.960
C07979=1067.539,102.710,427.057,172.747,27.237,154.960
C07980=1067.533,102.460,427.076,172.745,27.234,154.959
C07981=1067.528,102.212,427.095,172.744,27.231,154.959
C07982=1067.522,101.962,427.113,172.742,27.228,154.959
C07983=1067.516,101.712,427.132,172.741,27.225,154.958
C07984=1067.510,101.463,427.151,172.739,27.222,154.958
C07985=1067.505,101.215,427.170,172.738,27.220,154.957
C07986=1067.499,100.965,427.189,172.736,27.217,154.957
C07987=1067.493,100.716,427.208,172.735,27.215,154.957
C07988=1067.487,100.467,427.227,172.733,27.212,154.956
C07989=1067.480,100.217,427.245,172.732,27.209,154.956
C07990=1067.476,99.968,427.264,172.730,27.206,154.955
C07991=1067.469,99.719,427.282,172.729,27.203,154.955
C07992=1067.463,99.470,427.301,172.727,27.201,154.955
C07993=1067.457,99.220,427.320,172.725,27.198,154.954
C07994=1067.451,98.971,427.339,172.723,27.195,154.954
C07995=1067.446,98.723,427.358,172.722,27.192,154.954
C07996=1067.440,98.473,427.376,172.720,27.190,154.953
C07997=1067.434,98.223,427.395,172.719,27.187,154.953
C07998=1067.428,97.974,427.414,172.717,27.185,154.953
C07999=1067.422,97.726,427.432,172.716,27.182,154.952
C08000=1067.417,97.476,427.451,172.714,27.179,154.952
C08001=1067.410,97.226,427.470,172.713,27.176,154.951
C08002=1067.404,96.977,427.488,172.712,27.173,154.951
C08003=1067.399,96.729,427.507,172.710,27.171,154.951
C08004=1067.393,96.479,427.525,172.708,27.168,154.950
C08005=1067.387,96.229,427.544,172.707,27.166,154.950
C08006=1067.381,95.980,427.563,172.706,27.163,154.949
C08007=1067.376,95.731,427.581,172.704,27.160,154.949
C08008=1067.369,95.482,427.600,172.703,27.157,154.949
C08009=1067.364,95.232,427.619,172.701,27.155,154.948
C08010=1067.357,94.949,427.640,172.700,27.151,154.948
C08011=1067.351,94.666,427.661,172.697,27.148,154.947
C08012=1067.344,94.382,427.682,172.696,27.145,154.947
C08013=1067.337,94.099,427.703,172.694,27.142,154.947
C08014=1067.331,93.850,427.721,172.693,27.139,154.946
C08015=1067.326,93.601,427.740,172.691,27.137,154.946
C08016=1067.320,93.352,427.758,172.690,27.134,154.945
C08017=1067.314,93.102,427.777,172.688,27.131,154.945
C08018=1067.308,92.853,427.795,172.687,27.129,154.945
C08019=1067.302,92.604,427.814,172.685,27.126,154.944
C08020=1067.297,92.355,427.832,172.684,27.123,154.944
C08021=1067.291,92.106,427.850,172.682,27.120,154.943
C08022=1067.285,91.856,427.870,172.681,27.117,154.943
C08023=1067.280,91.607,427.887,172.680,27.115,154.943
C08024=1067.273,91.358,427.906,172.678,27.112,154.942
C08025=1067.268,91.108,427.924,172.677,27.109,154.942
C08026=1067.262,90.860,427.943,172.675,27.107,154.942
C08027=1067.256,90.610,427.961,172.674,27.104,154.941
C08028=1067.249,90.361,427.979,172.672,27.101,154.941
C08029=1067.244,90.112,427.998,172.671,27.098,154.940
C08030=1067.238,89.862,428.016,172.669,27.095,154.940
C08031=1067.232,89.613,428.035,172.668,27.093,154.940
C08032=1067.226,89.364,428.052,172.666,27.090,154.939
C08033=1067.220,89.114,428.070,172.665,27.088,154.939
C08034=1067.214,88.865,428.089,172.663,27.085,154.938
C08035=1067.209,88.616,428.107,172.662,27.082,154.938
C08036=1067.203,88.367,428.126,172.660,27.080,154.938
C08037=1067.196,88.117,428.144,172.659,27.077,154.937
C08038=1067.191,87.869,428.162,172.657,27.074,154.937
C08039=1067.184,87.619,428.180,172.656,27.071,154.937
C08040=1067.179,87.370,428.198,172.654,27.068,154.936
C08041=1067.173,87.120,428.217,172.653,27.066,154.936
C08042=1067.167,86.871,428.234,172.651,27.063,154.936
C08043=1067.161,86.622,428.253,172.650,27.061,154.935
C08044=1067.155,86.372,428.271,172.648,27.058,154.935
C08045=1067.149,86.124,428.289,172.647,27.055,154.934
C08046=1067.143,85.874,428.307,172.645,27.053,154.934
C08047=1067.137,85.624,428.325,172.644,27.050,154.934
C08048=1067.132,85.376,428.344,172.642,27.047,154.933
C08049=1067.126,85.126,428.362,172.641,27.044,154.933
C08050=1067.120,84.877,428.379,172.639,27.041,154.932
C08051=1067.114,84.628,428.398,172.638,27.039,154.932
C08052=1067.108,84.379,428.415,172.636,27.036,154.932
C08053=1067.102,84.129,428.433,172.635,27.033,154.931
C08054=1067.096,83.880,428.452,172.633,27.031,154.931
C08055=1067.090,83.631,428.470,172.632,27.028,154.931
C08056=1067.085,83.381,428.488,172.631,27.025,154.930
C08057=1067.080,83.132,428.506,172.629,27.022,154.930
C08058=1067.073,82.883,428.524,172.628,27.019,154.929
C08059=1067.068,82.634,428.542,172.626,27.017,154.929
C08060=1067.061,82.384,428.560,172.625,27.014,154.929
C08061=1067.056,82.135,428.577,172.623,27.011,154.928
C08062=1067.050,81.886,428.596,172.622,27.009,154.928
C08063=1067.044,81.637,428.614,172.620,27.006,154.927
C08064=1067.038,81.387,428.632,172.619,27.003,154.927
C08065=1067.032,81.138,428.649,172.617,27.000,154.927
C08066=1067.027,80.888,428.668,172.616,26.998,154.926
C08067=1067.021,80.639,428.686,172.614,26.995,154.926
C08068=1067.015,80.390,428.704,172.613,26.992,154.926
C08069=1067.010,80.141,428.721,172.611,26.989,154.925
C08070=1067.003,79.891,428.739,172.610,26.987,154.925
C08071=1066.998,79.642,428.757,172.608,26.984,154.924
C08072=1066.991,79.393,428.776,172.607,26.981,154.924
C08073=1066.986,79.144,428.793,172.606,26.978,154.924
C08074=1066.980,78.860,428.813,172.604,26.975,154.923
C08075=1066.973,78.577,428.833,172.602,26.972,154.923
C08076=1066.966,78.294,428.854,172.600,26.969,154.922
C08077=1066.959,78.011,428.874,172.599,26.966,154.922
C08078=1066.953,77.761,428.892,172.597,26.963,154.922
C08079=1066.948,77.512,428.909,172.596,26.960,154.921
C08080=1066.941,77.262,428.927,172.594,26.958,154.921
C08081=1066.936,77.013,428.945,172.593,26.955,154.920
C08082=1066.930,76.763,428.963,172.591,26.952,154.920
C08083=1066.924,76.515,428.980,172.590,26.950,154.920
C08084=1066.917,76.265,428.998,172.589,26.947,154.919
C08085=1066.912,76.016,429.015,172.587,26.945,154.919
C08086=1066.906,75.766,429.033,172.586,26.942,154.919
C08087=1066.900,75.517,429.051,172.584,26.939,154.918
C08088=1066.895,75.268,429.068,172.583,26.936,154.918
C08089=1066.889,75.018,429.086,172.581,26.933,154.917
C08090=1066.882,74.770,429.103,172.580,26.930,154.917
C08091=1066.876,74.520,429.121,172.578,26.928,154.917
C08092=1066.871,74.271,429.139,172.577,26.925,154.916
C08093=1066.865,74.021,429.157,172.575,26.922,154.916
C08094=1066.859,73.772,429.174,172.574,26.920,154.915
C08095=1066.853,73.522,429.192,172.572,26.917,154.915
C08096=1066.847,73.274,429.209,172.571,26.915,154.915
C08097=1066.841,73.025,429.227,172.569,26.912,154.914
C08098=1066.835,72.775,429.245,172.568,26.909,154.914
C08099=1066.830,72.526,429.262,172.566,26.906,154.914
C08100=1066.823,72.276,429.280,172.565,26.903,154.913
C08101=1066.817,72.027,429.297,172.565,26.901,154.913
C08102=1066.812,71.778,429.315,172.563,26.898,154.912
C08103=1066.806,71.529,429.333,172.562,26.896,154.912
C08104=1066.800,71.279,429.349,172.560,26.893,154.912
C08105=1066.794,71.029,429.367,172.559,26.890,154.911
C08106=1066.788,70.780,429.384,172.557,26.887,154.911
C08107=1066.782,70.531,429.402,172.556,26.884,154.910
C08108=1066.776,70.282,429.420,172.554,26.882,154.910
C08109=1066.771,70.033,429.437,172.553,26.879,154.910
C08110=1066.765,69.784,429.454,172.551,26.876,154.909
C08111=1066.759,69.533,429.472,172.550,26.873,154.909
C08112=1066.753,69.284,429.489,172.548,26.871,154.909
C08113=1066.746,69.035,429.506,172.547,26.868,154.908
C08114=1066.741,68.786,429.524,172.545,26.866,154.908
C08115=1066.735,68.537,429.542,172.544,26.863,154.908
C08116=1066.729,68.287,429.558,172.542,26.860,154.907
C08117=1066.723,68.038,429.576,172.541,26.857,154.907
C08118=1066.718,67.789,429.593,172.539,26.855,154.906
C08119=1066.711,67.539,429.611,172.538,26.852,154.906
C08120=1066.706,67.290,429.628,172.537,26.849,154.906
C08121=1066.700,67.041,429.645,172.535,26.846,154.905
C08122=1066.693,66.791,429.662,172.534,26.843,154.905
C08123=1066.688,66.542,429.680,172.532,26.841,154.905
C08124=1066.683,66.293,429.697,172.531,26.838,154.904
C08125=1066.676,66.043,429.714,172.529,26.836,154.904
C08126=1066.670,65.794,429.732,172.528,26.833,154.903
C08127=1066.664,65.545,429.748,172.526,26.830,154.903
C08128=1066.658,65.295,429.766,172.525,26.828,154.903
C08129=1066.653,65.046,429.784,172.523,26.825,154.902
C08130=1066.647,64.797,429.800,172.523,26.822,154.902
C08131=1066.641,64.547,429.818,172.521,26.819,154.901
C08132=1066.634,64.298,429.835,172.520,26.817,154.901
C08133=1066.629,64.048,429.852,172.518,26.814,154.901
C08134=1066.622,63.799,429.869,172.517,26.811,154.900
C08135=1066.616,63.550,429.886,172.516,26.809,154.900
C08136=1066.610,63.300,429.903,172.514,26.806,154.900
C08137=1066.604,63.051,429.920,172.513,26.803,154.899
C08138=1066.597,62.768,429.939,172.511,26.801,154.899
C08139=1066.590,62.484,429.959,172.509,26.797,154.899
C08140=1066.583,62.201,429.978,172.507,26.794,154.898
C08141=1066.577,61.918,429.997,172.506,26.791,154.898
C08142=1066.570,61.668,430.014,172.504,26.789,154.897
C08143=1066.564,61.419,430.031,172.503,26.786,154.897
C08144=1066.559,61.170,430.048,172.502,26.783,154.897
C08145=1066.552,60.920,430.066,172.500,26.780,154.896
C08146=1066.547,60.671,430.082,172.499,26.778,154.896
C08147=1066.541,60.422,430.099,172.497,26.775,154.896
C08148=1066.534,60.172,430.116,172.496,26.772,154.895
C08149=1066.528,59.923,430.134,172.494,26.770,154.895
C08150=1066.523,59.674,430.150,172.493,26.767,154.894
C08151=1066.516,59.425,430.167,172.491,26.765,154.894
C08152=1066.510,59.175,430.184,172.490,26.762,154.894
C08153=1066.505,58.925,430.200,172.488,26.759,154.893
C08154=1066.498,58.676,430.217,172.487,26.757,154.893
C08155=1066.492,58.426,430.234,172.485,26.754,154.893
C08156=1066.486,58.177,430.251,172.484,26.751,154.892
C08157=1066.480,57.928,430.268,172.483,26.749,154.892
C08158=1066.475,57.679,430.285,172.482,26.746,154.891
C08159=1066.468,57.429,430.302,172.480,26.743,154.891
C08160=1066.462,57.180,430.319,172.479,26.741,154.891
C08161=1066.457,56.931,430.336,172.477,26.738,154.890
C08162=1066.451,56.681,430.352,172.476,26.735,154.890
C08163=1066.444,56.432,430.369,172.475,26.732,154.890
C08164=1066.439,56.182,430.386,172.473,26.730,154.889
C08165=1066.432,55.933,430.403,172.472,26.727,154.889
C08166=1066.426,55.684,430.419,172.470,26.724,154.889
C08167=1066.421,55.435,430.436,172.469,26.722,154.888
C08168=1066.414,55.185,430.454,172.467,26.719,154.888
C08169=1066.408,54.936,430.470,172.466,26.716,154.887
C08170=1066.402,54.686,430.486,172.464,26.714,154.887
C08171=1066.397,54.437,430.504,172.463,26.711,154.887
C08172=1066.391,54.188,430.520,172.461,26.709,154.886
C08173=1066.385,53.938,430.536,172.460,26.706,154.886
C08174=1066.379,53.689,430.554,172.458,26.703,154.886
C08175=1066.373,53.439,430.570,172.457,26.700,154.885
C08176=1066.367,53.190,430.587,172.456,26.698,154.885
C08177=1066.361,52.941,430.603,172.454,26.695,154.885
C08178=1066.356,52.692,430.620,172.454,26.692,154.884
C08179=1066.350,52.442,430.637,172.452,26.689,154.884
C08180=1066.343,52.192,430.653,172.451,26.687,154.883
C08181=1066.337,51.943,430.670,172.449,26.684,154.883
C08182=1066.332,51.694,430.687,172.448,26.681,154.883
C08183=1066.326,51.445,430.703,172.446,26.679,154.882
C08184=1066.320,51.195,430.720,172.445,26.676,154.882
C08185=1066.314,50.946,430.736,172.443,26.673,154.882
C08186=1066.308,50.697,430.753,172.442,26.671,154.881
C08187=1066.302,50.447,430.770,172.441,26.668,154.881
C08188=1066.296,50.197,430.786,172.439,26.665,154.880
C08189=1066.291,49.948,430.803,172.438,26.663,154.880
C08190=1066.285,49.698,430.819,172.436,26.660,154.880
C08191=1066.279,49.449,430.836,172.435,26.657,154.879
C08192=1066.272,49.200,430.853,172.433,26.654,154.879
C08193=1066.266,48.951,430.869,172.432,26.651,154.879
C08194=1066.261,48.701,430.886,172.430,26.649,154.878
C08195=1066.255,48.452,430.902,172.429,26.646,154.878
C08196=1066.249,48.203,430.918,172.428,26.644,154.877
C08197=1066.243,47.953,430.935,172.427,26.641,154.877
C08198=1066.238,47.704,430.951,172.425,26.638,154.877
C08199=1066.232,47.455,430.968,172.424,26.636,154.876
C08200=1066.226,47.206,430.985,172.423,26.633,154.876
C08201=1066.220,46.956,431.001,172.421,26.630,154.876
C08202=1066.213,46.672,431.020,172.420,26.627,154.875
C08203=1066.207,46.388,431.039,172.417,26.623,154.875
C08204=1066.200,46.104,431.057,172.416,26.620,154.874
C08205=1066.193,45.822,431.076,172.415,26.618,154.874
C08206=1066.188,45.572,431.093,172.413,26.615,154.873
C08207=1066.182,45.323,431.109,172.412,26.612,154.873
C08208=1066.176,45.073,431.125,172.410,26.609,154.873
C08209=1066.170,44.824,431.141,172.409,26.607,154.872
C08210=1066.164,44.575,431.158,172.407,26.604,154.872
C08211=1066.158,44.325,431.174,172.406,26.601,154.872
C08212=1066.153,44.076,431.191,172.405,26.598,154.871
C08213=1066.147,43.826,431.207,172.403,26.595,154.871
C08214=1066.141,43.577,431.223,172.402,26.593,154.871
C08215=1066.135,43.328,431.240,172.401,26.591,154.870
C08216=1066.129,43.078,431.256,172.400,26.588,154.870
C08217=1066.123,42.829,431.272,172.398,26.585,154.869
C08218=1066.117,42.580,431.288,172.397,26.583,154.869
C08219=1066.111,42.329,431.304,172.395,26.580,154.869
C08220=1066.105,42.079,431.321,172.394,26.577,154.868
C08221=1066.099,41.830,431.337,172.392,26.575,154.868
C08222=1066.093,41.581,431.353,172.391,26.572,154.868
C08223=1066.087,41.331,431.369,172.389,26.569,154.867
C08224=1066.081,41.082,431.386,172.388,26.567,154.867
C08225=1066.075,40.833,431.402,172.387,26.564,154.867
C08226=1066.069,40.583,431.418,172.385,26.561,154.866
C08227=1066.063,40.334,431.434,172.384,26.558,154.866
C08228=1066.058,40.085,431.451,172.382,26.556,154.865
C08229=1066.052,39.835,431.466,172.381,26.553,154.865
C08230=1066.047,39.586,431.482,172.379,26.550,154.865
C08231=1066.041,39.337,431.498,172.378,26.548,154.864
C08232=1066.034,39.088,431.514,172.376,26.545,154.864
C08233=1066.028,38.838,431.530,172.376,26.542,154.864
C08234=1066.022,38.589,431.546,172.374,26.539,154.863
C08235=1066.016,38.339,431.562,172.373,26.537,154.863
C08236=1066.010,38.090,431.578,172.372,26.534,154.863
C08237=1066.004,37.840,431.595,172.370,26.531,154.862
C08238=1065.998,37.591,431.611,172.369,26.529,154.862
C08239=1065.993,37.342,431.627,172.367,26.526,154.861
C08240=1065.987,37.092,431.643,172.366,26.523,154.861
C08241=1065.980,36.843,431.658,172.364,26.521,154.861
C08242=1065.974,36.593,431.674,172.363,26.518,154.860
C08243=1065.968,36.344,431.691,172.361,26.516,154.860
C08244=1065.963,36.094,431.706,172.360,26.513,154.860
C08245=1065.956,35.845,431.722,172.358,26.510,154.859
C08246=1065.950,35.596,431.738,172.357,26.508,154.859
C08247=1065.944,35.346,431.754,172.355,26.505,154.859
C08248=1065.938,35.096,431.770,172.354,26.502,154.858
C08249=1065.932,34.847,431.786,172.353,26.500,154.858
C08250=1065.926,34.598,431.802,172.351,26.497,154.858
C08251=1065.920,34.348,431.817,172.351,26.494,154.857
C08252=1065.914,34.099,431.834,172.349,26.492,154.857
C08253=1065.907,33.850,431.849,172.348,26.489,154.856
C08254=1065.902,33.600,431.865,172.346,26.487,154.856
C08255=1065.896,33.351,431.881,172.345,26.484,154.856
C08256=1065.891,33.101,431.896,172.343,26.481,154.855
C08257=1065.884,32.852,431.912,172.342,26.479,154.855
C08258=1065.878,32.603,431.928,172.340,26.476,154.855
C08259=1065.873,32.353,431.944,172.339,26.473,154.854
C08260=1065.867,32.103,431.960,172.337,26.471,154.854
C08261=1065.860,31.854,431.976,172.336,26.468,154.854
C08262=1065.854,31.604,431.991,172.335,26.465,154.853
C08263=1065.848,31.355,432.008,172.333,26.463,154.853
C08264=1065.843,31.106,432.022,172.332,26.460,154.853
C08265=1065.837,30.857,432.038,172.330,26.458,154.852
C08266=1065.829,30.573,432.056,172.329,26.454,154.852
C08267=1065.823,30.289,432.075,172.327,26.451,154.851
C08268=1065.816,30.005,432.093,172.326,26.449,154.851
C08269=1065.810,29.722,432.110,172.325,26.446,154.851
C08270=1065.804,29.472,432.126,172.323,26.443,154.850
C08271=1065.798,29.223,432.141,172.322,26.441,154.850
C08272=1065.792,28.973,432.157,172.320,26.438,154.850
C08273=1065.786,28.723,432.173,172.319,26.435,154.849
C08274=1065.780,28.475,432.188,172.317,26.433,154.849
C08275=1065.774,28.225,432.203,172.316,26.430,154.849
C08276=1065.767,27.976,432.219,172.314,26.427,154.848
C08277=1065.762,27.726,432.235,172.313,26.425,154.848
C08278=1065.756,27.477,432.251,172.312,26.422,154.848
C08279=1065.750,27.227,432.266,172.310,26.419,154.847
C08280=1065.744,26.978,432.282,172.309,26.417,154.847
C08281=1065.738,26.729,432.297,172.307,26.414,154.847
C08282=1065.732,26.479,432.313,172.306,26.411,154.846
C08283=1065.725,26.230,432.328,172.304,26.409,154.846
C08284=1065.720,25.980,432.343,172.303,26.406,154.845
C08285=1065.713,25.731,432.359,172.301,26.404,154.845
C08286=1065.707,25.481,432.375,172.300,26.401,154.845
C08287=1065.701,25.232,432.390,172.298,26.399,154.845
C08288=1065.696,24.982,432.405,172.298,26.396,154.844
C08289=1065.689,24.733,432.420,172.297,26.393,154.844
C08290=1065.683,24.483,432.437,172.295,26.391,154.843
C08291=1065.677,24.234,432.452,172.294,26.388,154.843
C08292=1065.672,23.984,432.467,172.292,26.386,154.843
C08293=1065.665,23.735,432.482,172.291,26.383,154.842
C08294=1065.660,23.485,432.498,172.289,26.381,154.842
C08295=1065.653,23.236,432.513,172.288,26.378,154.842
C08296=1065.647,22.986,432.529,172.286,26.375,154.841
C08297=1065.642,22.737,432.544,172.285,26.373,154.841
C08298=1065.636,22.487,432.559,172.283,26.370,154.841
C08299=1065.629,22.238,432.575,172.282,26.367,154.840
C08300=1065.624,21.988,432.591,172.281,26.365,154.840
C08301=1065.618,21.740,432.605,172.279,26.362,154.840
C08302=1065.612,21.490,432.621,172.278,26.359,154.839
C08303=1065.605,21.241,432.636,172.276,26.357,154.839
C08304=1065.599,20.991,432.651,172.275,26.354,154.839
C08305=1065.594,20.742,432.666,172.273,26.351,154.838
C08306=1065.587,20.493,432.682,172.273,26.349,154.838
C08307=1065.582,20.243,432.698,172.271,26.346,154.838
C08308=1065.575,19.993,432.713,172.270,26.344,154.837
C08309=1065.570,19.744,432.728,172.268,26.341,154.837
C08310=1065.564,19.494,432.743,172.267,26.339,154.837
C08311=1065.557,19.245,432.758,172.265,26.336,154.836
C08312=1065.552,18.995,432.774,172.264,26.334,154.836
C08313=1065.546,18.746,432.788,172.263,26.331,154.836
C08314=1065.539,18.496,432.803,172.261,26.329,154.835
C08315=1065.534,18.246,432.819,172.260,26.326,154.835
C08316=1065.527,17.997,432.834,172.258,26.323,154.835
C08317=1065.521,17.748,432.849,172.257,26.321,154.834
C08318=1065.516,17.498,432.865,172.255,26.318,154.834
C08319=1065.509,17.249,432.880,172.254,26.315,154.834
C08320=1065.503,17.000,432.894,172.252,26.313,154.833
C08321=1065.498,16.750,432.910,172.251,26.310,154.833
C08322=1065.491,16.500,432.925,172.249,26.308,154.833
C08323=1065.485,16.251,432.940,172.248,26.305,154.832
C08324=1065.480,16.001,432.955,172.246,26.303,154.832
C08325=1065.473,15.752,432.971,172.245,26.300,154.832
C08326=1065.467,15.503,432.985,172.245,26.298,154.831
C08327=1065.461,15.254,433.000,172.243,26.295,154.831
C08328=1065.455,15.004,433.016,172.242,26.293,154.831
C08329=1065.449,14.754,433.031,172.240,26.290,154.830
C08330=1065.442,14.472,433.047,172.238,26.287,154.830
C08331=1065.436,14.190,433.064,172.236,26.284,154.830
C08332=1065.429,13.908,433.081,172.235,26.281,154.829
C08333=1065.422,13.624,433.098,172.234,26.279,154.829
C08334=1065.416,13.376,433.113,172.232,26.276,154.828
C08335=1065.410,13.126,433.128,172.231,26.273,154.828
C08336=1065.404,12.876,433.143,172.229,26.271,154.828
C08337=1065.398,12.627,433.157,172.228,26.268,154.827
C08338=1065.391,12.378,433.172,172.226,26.266,154.827
C08339=1065.385,12.128,433.187,172.225,26.264,154.827
C08340=1065.379,11.879,433.202,172.223,26.261,154.827
C08341=1065.373,11.629,433.217,172.222,26.258,154.826
C08342=1065.366,11.380,433.232,172.220,26.256,154.826
C08343=1065.361,11.131,433.246,172.219,26.253,154.826
C08344=1065.355,10.881,433.262,172.217,26.251,154.825
C08345=1065.349,10.631,433.277,172.216,26.248,154.825
C08346=1065.343,10.382,433.291,172.215,26.246,154.825
C08347=1065.336,10.132,433.306,172.213,26.243,154.824
C08348=1065.330,9.883,433.321,172.212,26.240,154.824
C08349=1065.325,9.633,433.335,172.210,26.238,154.824
C08350=1065.318,9.384,433.350,172.210,26.236,154.823
C08351=1065.312,9.134,433.365,172.208,26.233,154.823
C08352=1065.306,8.885,433.380,172.207,26.231,154.823
C08353=1065.300,8.635,433.395,172.205,26.229,154.822
C08354=1065.294,8.386,433.409,172.204,26.226,154.822
C08355=1065.288,8.137,433.424,172.202,26.223,154.822
C08356=1065.281,7.886,433.438,172.201,26.221,154.821
C08357=1065.276,7.637,433.453,172.199,26.218,154.821
C08358=1065.269,7.388,433.468,172.198,26.216,154.821
C08359=1065.263,7.139,433.482,172.196,26.213,154.820
C08360=1065.258,6.889,433.498,172.195,26.211,154.820
C08361=1065.252,6.639,433.512,172.193,26.208,154.820
C08362=1065.246,6.390,433.527,172.192,26.206,154.820
C08363=1065.240,6.140,433.542,172.191,26.203,154.819
C08364=1065.234,5.891,433.556,172.189,26.200,154.819
C08365=1065.227,5.641,433.571,172.188,26.198,154.819
C08366=1065.222,5.392,433.585,172.186,26.196,154.818
C08367=1065.216,5.142,433.600,172.185,26.193,154.818
C08368=1065.209,4.892,433.615,172.183,26.191,154.818
C08369=1065.203,4.644,433.630,172.182,26.188,154.817
C08370=1065.197,4.393,433.644,172.180,26.185,154.817
C08371=1065.192,4.144,433.658,172.179,26.183,154.817
C08372=1065.185,3.895,433.673,172.177,26.181,154.816
C08373=1065.180,3.645,433.687,172.176,26.178,154.816
C08374=1065.173,3.395,433.702,172.174,26.176,154.816
C08375=1065.168,3.146,433.717,172.174,26.173,154.815
C08376=1065.161,2.897,433.732,172.172,26.171,154.815
C08377=1065.156,2.647,433.746,172.171,26.168,154.815
C08378=1065.149,2.398,433.760,172.170,26.165,154.814
C08379=1065.144,2.149,433.775,172.168,26.163,154.814
C08380=1065.137,1.898,433.789,172.167,26.161,154.814
C08381=1065.132,1.649,433.804,172.165,26.158,154.814
C08382=1065.125,1.400,433.819,172.164,26.156,154.813
C08383=1065.120,1.150,433.833,172.162,26.153,154.813
C08384=1065.113,0.900,433.848,172.161,26.150,154.813
C08385=1065.108,0.651,433.861,172.159,26.148,154.812
C08386=1065.102,0.401,433.876,172.158,26.146,154.812
C08387=1065.096,0.152,433.891,172.156,26.143,154.812
C08388=1065.090,-0.097,433.905,172.155,26.141,154.811
C08389=1065.084,-0.347,433.920,172.153,26.138,154.811
C08390=1065.078,-0.596,433.934,172.152,26.135,154.811
C08391=1065.072,-0.846,433.949,172.151,26.133,154.810
C08392=1065.066,-1.095,433.962,172.149,26.131,154.810
C08393=1065.059,-1.345,433.977,172.148,26.128,154.810
C08394=1065.054,-1.625,433.994,172.146,26.125,154.809
C08395=1065.047,-1.906,434.009,172.145,26.123,154.809
C08396=1065.040,-2.186,434.025,172.143,26.120,154.809
C08397=1065.033,-2.466,434.041,172.141,26.117,154.808
C08398=1065.027,-2.716,434.056,172.140,26.114,154.808
C08399=1065.022,-2.965,434.070,172.138,26.111,154.808
C08400=1065.015,-3.215,434.084,172.137,26.109,154.807
C08401=1065.010,-3.464,434.099,172.135,26.107,154.807
C08402=1065.003,-3.714,434.113,172.134,26.104,154.807
C08403=1064.997,-3.963,434.127,172.132,26.102,154.807
C08404=1064.992,-4.213,434.141,172.131,26.099,154.806
C08405=1064.985,-4.462,434.156,172.130,26.097,154.806
C08406=1064.979,-4.712,434.169,172.129,26.095,154.806
C08407=1064.973,-4.962,434.184,172.127,26.092,154.805
C08408=1064.967,-5.211,434.198,172.126,26.090,154.805
C08409=1064.960,-5.461,434.212,172.124,26.088,154.805
C08410=1064.955,-5.710,434.226,172.123,26.085,154.804
C08411=1064.948,-5.960,434.241,172.121,26.083,154.804
C08412=1064.942,-6.209,434.255,172.120,26.080,154.804
C08413=1064.936,-6.458,434.268,172.118,26.078,154.804
C08414=1064.930,-6.709,434.283,172.117,26.076,154.803
C08415=1064.924,-6.957,434.297,172.115,26.073,154.803
C08416=1064.918,-7.208,434.311,172.114,26.070,154.803
C08417=1064.912,-7.457,434.325,172.113,26.068,154.802
C08418=1064.906,-7.706,434.339,172.111,26.066,154.802
C08419=1064.900,-7.956,434.353,172.110,26.063,154.802
C08420=1064.894,-8.206,434.367,172.108,26.061,154.802
C08421=1064.887,-8.455,434.381,172.107,26.059,154.801
C08422=1064.882,-8.705,434.395,172.105,26.056,154.801
C08423=1064.876,-8.954,434.409,172.104,26.054,154.801
C08424=1064.869,-9.203,434.423,172.102,26.051,154.800
C08425=1064.864,-9.453,434.437,172.101,26.049,154.800
C08426=1064.857,-9.703,434.451,172.099,26.047,154.800
C08427=1064.851,-9.953,434.465,172.098,26.044,154.800
C08428=1064.845,-10.202,434.479,172.096,26.042,154.799
C08429=1064.839,-10.451,434.493,172.095,26.039,154.799
C08430=1064.833,-10.701,434.507,172.093,26.037,154.799
C08431=1064.827,-10.950,434.521,172.092,26.034,154.798
C08432=1064.821,-11.200,434.535,172.090,26.032,154.798
C08433=1064.815,-11.450,434.549,172.089,26.030,154.798
C08434=1064.809,-11.699,434.562,172.087,26.027,154.798
C08435=1064.803,-11.949,434.576,172.086,26.025,154.797
C08436=1064.797,-12.198,434.591,172.084,26.022,154.797
C08437=1064.791,-12.447,434.604,172.083,26.020,154.797
C08438=1064.785,-12.697,434.618,172.081,26.018,154.796
C08439=1064.779,-12.947,434.632,172.080,26.015,154.796
C08440=1064.773,-13.196,434.646,172.078,26.013,154.796
C08441=1064.767,-13.445,434.660,172.077,26.011,154.796
C08442=1064.760,-13.695,434.674,172.075,26.008,154.795
C08443=1064.755,-13.945,434.688,172.074,26.006,154.795
C08444=1064.750,-14.195,434.701,172.073,26.003,154.795
C08445=1064.743,-14.444,434.715,172.071,26.001,154.794
C08446=1064.737,-14.694,434.729,172.070,25.998,154.794
C08447=1064.731,-14.943,434.742,172.068,25.996,154.794
C08448=1064.726,-15.193,434.756,172.067,25.994,154.794
C08449=1064.718,-15.442,434.770,172.065,25.991,154.793
C08450=1064.713,-15.692,434.784,172.064,25.989,154.793
C08451=1064.707,-15.941,434.798,172.062,25.987,154.793
C08452=1064.700,-16.191,434.811,172.061,25.984,154.793
C08453=1064.694,-16.441,434.825,172.059,25.982,154.792
C08454=1064.688,-16.690,434.838,172.058,25.980,154.792
C08455=1064.683,-16.939,434.852,172.056,25.978,154.792
C08456=1064.676,-17.189,434.866,172.055,25.975,154.791
C08457=1064.670,-17.439,434.879,172.053,25.973,154.791
C08458=1064.663,-17.717,434.894,172.052,25.971,154.791
C08459=1064.656,-17.996,434.909,172.050,25.968,154.791
C08460=1064.649,-18.275,434.925,172.049,25.965,154.790
C08461=1064.643,-18.554,434.940,172.046,25.963,154.790
C08462=1064.637,-18.803,434.954,172.045,25.960,154.790
C08463=1064.630,-19.053,434.967,172.043,25.958,154.790
C08464=1064.624,-19.302,434.980,172.042,25.956,154.789
C08465=1064.619,-19.552,434.994,172.041,25.953,154.789
C08466=1064.612,-19.801,435.008,172.039,25.951,154.789
C08467=1064.606,-20.051,435.021,172.038,25.949,154.788
C08468=1064.600,-20.301,435.035,172.036,25.946,154.788
C08469=1064.594,-20.550,435.048,172.035,25.944,154.788
C08470=1064.588,-20.800,435.062,172.033,25.942,154.788
C08471=1064.582,-21.049,435.075,172.032,25.939,154.787
C08472=1064.575,-21.299,435.089,172.030,25.937,154.787
C08473=1064.570,-21.548,435.103,172.029,25.935,154.787
C08474=1064.564,-21.798,435.116,172.027,25.932,154.787
C08475=1064.557,-22.047,435.129,172.027,25.930,154.786
C08476=1064.552,-22.297,435.143,172.025,25.928,154.786
C08477=1064.546,-22.547,435.156,172.024,25.926,154.786
C08478=1064.539,-22.796,435.170,172.022,25.924,154.786
C08479=1064.534,-23.046,435.183,172.020,25.922,154.785
C08480=1064.528,-23.295,435.197,172.019,25.919,154.785
C08481=1064.521,-23.545,435.210,172.017,25.917,154.785
C08482=1064.515,-23.794,435.223,172.016,25.915,154.785
C08483=1064.509,-24.044,435.237,172.015,25.912,154.784
C08484=1064.503,-24.294,435.250,172.013,25.910,154.784
C08485=1064.497,-24.543,435.263,172.012,25.908,154.784
C08486=1064.491,-24.793,435.277,172.009,25.905,154.784
C08487=1064.485,-25.042,435.290,172.008,25.903,154.783
C08488=1064.479,-25.291,435.304,172.006,25.900,154.783
C08489=1064.474,-25.542,435.317,172.005,25.898,154.783
C08490=1064.467,-25.791,435.330,172.003,25.896,154.782
C08491=1064.461,-26.041,435.344,172.002,25.893,154.782
C08492=1064.455,-26.290,435.358,172.000,25.892,154.782
C08493=1064.449,-26.540,435.371,171.999,25.889,154.782
C08494=1064.443,-26.789,435.383,171.997,25.887,154.781
C08495=1064.437,-27.039,435.397,171.996,25.885,154.781
C08496=1064.431,-27.288,435.410,171.994,25.882,154.781
C08497=1064.424,-27.539,435.423,171.993,25.880,154.781
C08498=1064.419,-27.788,435.437,171.991,25.878,154.781
C08499=1064.413,-28.037,435.450,171.990,25.876,154.780
C08500=1064.406,-28.287,435.463,171.988,25.873,154.780
C08501=1064.401,-28.537,435.476,171.987,25.871,154.780
C08502=1064.394,-28.786,435.489,171.985,25.869,154.780
C08503=1064.388,-29.035,435.502,171.984,25.867,154.779
C08504=1064.382,-29.285,435.515,171.982,25.865,154.779
C08505=1064.375,-29.535,435.529,171.981,25.862,154.779
C08506=1064.369,-29.784,435.542,171.979,25.860,154.779
C08507=1064.363,-30.034,435.554,171.977,25.858,154.778
C08508=1064.357,-30.283,435.568,171.976,25.856,154.778
C08509=1064.351,-30.533,435.581,171.974,25.854,154.778
C08510=1064.345,-30.782,435.593,171.973,25.851,154.778
C08511=1064.339,-31.032,435.607,171.971,25.849,154.777
C08512=1064.334,-31.282,435.620,171.970,25.847,154.777
C08513=1064.327,-31.531,435.633,171.968,25.845,154.777
C08514=1064.321,-31.780,435.646,171.967,25.843,154.777
C08515=1064.315,-32.031,435.659,171.965,25.841,154.777
C08516=1064.308,-32.280,435.673,171.964,25.838,154.776
C08517=1064.302,-32.530,435.685,171.962,25.836,154.776
C08518=1064.296,-32.779,435.698,171.961,25.834,154.776
C08519=1064.290,-33.029,435.711,171.959,25.832,154.776
C08520=1064.284,-33.279,435.724,171.958,25.830,154.775
C08521=1064.278,-33.529,435.737,171.956,25.827,154.775
C08522=1064.271,-33.806,435.752,171.955,25.825,154.775
C08523=1064.265,-34.084,435.766,171.953,25.823,154.774
C08524=1064.258,-34.361,435.781,171.951,25.820,154.774
C08525=1064.251,-34.639,435.795,171.949,25.818,154.774
C08526=1064.245,-34.889,435.807,171.948,25.816,154.774
C08527=1064.239,-35.139,435.820,171.946,25.813,154.774
C08528=1064.233,-35.388,435.833,171.945,25.811,154.773
C08529=1064.227,-35.638,435.846,171.943,25.809,154.773
C08530=1064.221,-35.887,435.859,171.942,25.807,154.773
C08531=1064.215,-36.137,435.872,171.940,25.805,154.773
C08532=1064.209,-36.386,435.885,171.939,25.802,154.772
C08533=1064.203,-36.636,435.897,171.937,25.801,154.772
C08534=1064.197,-36.886,435.911,171.936,25.798,154.772
C08535=1064.191,-37.135,435.923,171.934,25.796,154.772
C08536=1064.184,-37.385,435.936,171.933,25.794,154.772
C08537=1064.179,-37.635,435.949,171.931,25.792,154.771
C08538=1064.173,-37.884,435.962,171.930,25.789,154.771
C08539=1064.166,-38.134,435.975,171.928,25.788,154.771
C08540=1064.161,-38.384,435.987,171.927,25.785,154.771
C08541=1064.155,-38.633,436.000,171.925,25.783,154.770
C08542=1064.148,-38.883,436.013,171.924,25.781,154.770
C08543=1064.143,-39.133,436.026,171.922,25.779,154.770
C08544=1064.136,-39.382,436.039,171.921,25.777,154.770
C08545=1064.130,-39.632,436.052,171.919,25.775,154.770
C08546=1064.124,-39.881,436.064,171.917,25.773,154.769
C08547=1064.118,-40.131,436.077,171.916,25.771,154.769
C08548=1064.112,-40.381,436.089,171.914,25.769,154.769
C08549=1064.106,-40.630,436.102,171.913,25.767,154.769
C08550=1064.099,-40.880,436.115,171.911,25.765,154.769
C08551=1064.093,-41.129,436.127,171.910,25.762,154.768
C08552=1064.087,-41.379,436.140,171.908,25.761,154.768
C08553=1064.081,-41.629,436.152,171.907,25.758,154.768
C08554=1064.075,-41.878,436.166,171.905,25.757,154.768
C08555=1064.068,-42.128,436.177,171.904,25.754,154.767
C08556=1064.062,-42.378,436.190,171.902,25.753,154.767
C08557=1064.056,-42.628,436.203,171.901,25.750,154.767
C08558=1064.050,-42.877,436.216,171.898,25.748,154.767
C08559=1064.043,-43.126,436.228,171.897,25.746,154.767
C08560=1064.038,-43.376,436.240,171.895,25.744,154.767
C08561=1064.032,-43.625,436.253,171.893,25.742,154.766
C08562=1064.026,-43.875,436.266,171.892,25.740,154.766
C08563=1064.020,-44.125,436.278,171.890,25.738,154.766
C08564=1064.014,-44.374,436.290,171.889,25.736,154.766
C08565=1064.008,-44.624,436.303,171.887,25.733,154.765
C08566=1064.002,-44.874,436.315,171.886,25.732,154.765
C08567=1063.995,-45.123,436.328,171.884,25.729,154.765
C08568=1063.989,-45.373,436.341,171.883,25.728,154.765
C08569=1063.983,-45.623,436.353,171.881,25.725,154.765
C08570=1063.978,-45.872,436.365,171.880,25.723,154.765
C08571=1063.971,-46.121,436.377,171.878,25.721,154.764
C08572=1063.965,-46.371,436.390,171.876,25.719,154.764
C08573=1063.959,-46.621,436.403,171.875,25.718,154.764
C08574=1063.953,-46.870,436.416,171.873,25.715,154.764
C08575=1063.946,-47.120,436.428,171.872,25.713,154.764
C08576=1063.940,-47.370,436.440,171.870,25.711,154.763
C08577=1063.935,-47.619,436.452,171.869,25.709,154.763
C08578=1063.928,-47.869,436.464,171.867,25.707,154.763
C08579=1063.923,-48.119,436.477,171.866,25.705,154.763
C08580=1063.917,-48.368,436.490,171.864,25.703,154.763
C08581=1063.911,-48.618,436.502,171.863,25.701,154.762
C08582=1063.905,-48.867,436.514,171.861,25.699,154.762
C08583=1063.899,-49.117,436.526,171.860,25.697,154.762
C08584=1063.893,-49.367,436.539,171.858,25.695,154.762
C08585=1063.886,-49.617,436.551,171.856,25.693,154.762
C08586=1063.879,-49.894,436.565,171.854,25.691,154.761
C08587=1063.873,-50.173,436.579,171.852,25.688,154.761
C08588=1063.867,-50.451,436.592,171.851,25.687,154.761
C08589=1063.859,-50.730,436.606,171.849,25.684,154.761
C08590=1063.853,-50.980,436.618,171.848,25.683,154.761
C08591=1063.847,-51.229,436.630,171.846,25.681,154.760
C08592=1063.841,-51.479,436.642,171.844,25.678,154.760
C08593=1063.834,-51.728,436.654,171.842,25.676,154.760
C08594=1063.828,-51.978,436.666,171.841,25.675,154.760
C08595=1063.822,-52.228,436.679,171.839,25.673,154.760
C08596=1063.815,-52.477,436.691,171.837,25.671,154.760
C08597=1063.809,-52.727,436.703,171.836,25.669,154.760
C08598=1063.803,-52.976,436.715,171.834,25.667,154.759
C08599=1063.797,-53.226,436.727,171.833,25.665,154.759
C08600=1063.791,-53.475,436.739,171.831,25.663,154.759
C08601=1063.784,-53.725,436.751,171.830,25.662,154.759
C08602=1063.778,-53.975,436.764,171.828,25.660,154.759
C08603=1063.772,-54.224,436.775,171.826,25.657,154.758
C08604=1063.766,-54.474,436.787,171.825,25.656,154.758
C08605=1063.760,-54.724,436.799,171.823,25.654,154.758
C08606=1063.753,-54.973,436.811,171.822,25.652,154.758
C08607=1063.747,-55.223,436.823,171.820,25.650,154.758
C08608=1063.741,-55.472,436.835,171.818,25.649,154.758
C08609=1063.735,-55.722,436.847,171.817,25.647,154.758
C08610=1063.729,-55.972,436.859,171.815,25.644,154.757
C08611=1063.722,-56.222,436.871,171.814,25.643,154.757
C08612=1063.716,-56.471,436.883,171.812,25.641,154.757
C08613=1063.710,-56.721,436.895,171.811,25.639,154.757
C08614=1063.704,-56.970,436.907,171.809,25.637,154.757
C08615=1063.697,-57.220,436.919,171.807,25.636,154.757
C08616=1063.691,-57.470,436.931,171.805,25.633,154.756
C08617=1063.685,-57.719,436.943,171.803,25.632,154.756
C08618=1063.679,-57.969,436.955,171.802,25.630,154.756
C08619=1063.673,-58.219,436.967,171.800,25.628,154.756
C08620=1063.667,-58.469,436.978,171.799,25.626,154.756
C08621=1063.660,-58.718,436.990,171.797,25.624,154.756
C08622=1063.655,-58.967,437.003,171.795,25.622,154.756
C08623=1063.648,-59.217,437.015,171.794,25.620,154.755
C08624=1063.642,-59.467,437.025,171.792,25.619,154.755
C08625=1063.636,-59.716,437.038,171.791,25.617,154.755
C08626=1063.630,-59.966,437.050,171.789,25.615,154.755
C08627=1063.623,-60.216,437.061,171.787,25.613,154.755
C08628=1063.618,-60.465,437.073,171.786,25.612,154.755
C08629=1063.611,-60.715,437.085,171.784,25.610,154.755
C08630=1063.605,-60.965,437.097,171.783,25.608,154.754
C08631=1063.600,-61.214,437.109,171.781,25.606,154.754
C08632=1063.593,-61.464,437.121,171.780,25.604,154.754
C08633=1063.587,-61.714,437.132,171.778,25.602,154.754
C08634=1063.581,-61.963,437.144,171.776,25.600,154.754
C08635=1063.575,-62.213,437.156,171.775,25.599,154.754
C08636=1063.568,-62.463,437.167,171.773,25.597,154.753
C08637=1063.562,-62.712,437.179,171.772,25.595,154.753
C08638=1063.556,-62.962,437.191,171.770,25.593,154.753
C08639=1063.550,-63.212,437.203,171.768,25.591,154.753
C08640=1063.544,-63.461,437.214,171.766,25.589,154.753
C08641=1063.538,-63.711,437.226,171.764,25.588,154.753
C08642=1063.532,-63.960,437.238,171.763,25.586,154.753
C08643=1063.526,-64.210,437.250,171.761,25.584,154.752
C08644=1063.519,-64.460,437.261,171.760,25.582,154.752
C08645=1063.514,-64.709,437.273,171.758,25.581,154.752
C08646=1063.508,-64.959,437.284,171.756,25.579,154.752
C08647=1063.502,-65.208,437.296,171.755,25.577,154.752
C08648=1063.496,-65.459,437.308,171.753,25.575,154.752
C08649=1063.489,-65.708,437.320,171.752,25.573,154.752
C08650=1063.483,-65.988,437.333,171.750,25.572,154.751
C08651=1063.476,-66.267,437.346,171.747,25.570,154.751
C08652=1063.469,-66.547,437.359,171.746,25.568,154.751
C08653=1063.462,-66.826,437.372,171.744,25.565,154.751
C08654=1063.456,-67.077,437.383,171.743,25.564,154.751
C08655=1063.450,-67.325,437.395,171.741,25.562,154.751
C08656=1063.444,-67.576,437.407,171.740,25.561,154.751
C08657=1063.438,-67.825,437.418,171.738,25.559,154.751
C08658=1063.432,-68.075,437.429,171.736,25.557,154.750
C08659=1063.426,-68.324,437.441,171.735,25.555,154.750
C08660=1063.420,-68.574,437.452,171.733,25.554,154.750
C08661=1063.414,-68.825,437.464,171.731,25.551,154.750
C08662=1063.408,-69.073,437.476,171.729,25.550,154.750
C08663=1063.402,-69.324,437.487,171.727,25.548,154.750
C08664=1063.396,-69.572,437.498,171.726,25.546,154.750
C08665=1063.390,-69.823,437.510,171.724,25.544,154.749
C08666=1063.384,-70.072,437.522,171.723,25.543,154.749
C08667=1063.378,-70.322,437.533,171.721,25.541,154.749
C08668=1063.372,-70.572,437.544,171.719,25.540,154.749
C08669=1063.365,-70.821,437.556,171.718,25.538,154.749
C08670=1063.360,-71.071,437.567,171.716,25.536,154.749
C08671=1063.354,-71.321,437.579,171.715,25.534,154.749
C08672=1063.348,-71.570,437.590,171.713,25.532,154.749
C08673=1063.342,-71.820,437.602,171.711,25.531,154.748
C08674=1063.336,-72.069,437.613,171.710,25.529,154.748
C08675=1063.331,-72.319,437.625,171.708,25.528,154.748
C08676=1063.324,-72.569,437.636,171.706,25.526,154.748
C08677=1063.318,-72.818,437.647,171.705,25.524,154.748
C08678=1063.312,-73.068,437.659,171.703,25.522,154.748
C08679=1063.306,-73.318,437.670,171.702,25.521,154.748
C08680=1063.300,-73.568,437.681,171.700,25.519,154.748
C08681=1063.294,-73.817,437.693,171.699,25.517,154.747
C08682=1063.288,-74.067,437.704,171.697,25.516,154.747
C08683=1063.282,-74.317,437.715,171.694,25.514,154.747
C08684=1063.276,-74.566,437.727,171.693,25.512,154.747
C08685=1063.270,-74.816,437.738,171.691,25.511,154.747
C08686=1063.264,-75.066,437.749,171.689,25.509,154.747
C08687=1063.258,-75.315,437.760,171.688,25.507,154.747
C08688=1063.251,-75.565,437.772,171.686,25.506,154.747
C08689=1063.245,-75.814,437.783,171.684,25.504,154.747
C08690=1063.240,-76.064,437.794,171.683,25.502,154.747
C08691=1063.233,-76.314,437.804,171.681,25.501,154.747
C08692=1063.227,-76.563,437.815,171.680,25.499,154.746
C08693=1063.220,-76.813,437.827,171.678,25.498,154.746
C08694=1063.215,-77.062,437.838,171.676,25.496,154.746
C08695=1063.208,-77.313,437.849,171.675,25.495,154.746
C08696=1063.202,-77.562,437.860,171.673,25.493,154.746
C08697=1063.196,-77.812,437.871,171.671,25.492,154.746
C08698=1063.190,-78.062,437.882,171.670,25.490,154.746
C08699=1063.184,-78.311,437.894,171.668,25.489,154.746
C08700=1063.178,-78.561,437.905,171.666,25.487,154.746
C08701=1063.172,-78.810,437.916,171.665,25.485,154.746
C08702=1063.166,-79.060,437.927,171.663,25.484,154.745
C08703=1063.160,-79.310,437.938,171.661,25.482,154.745
C08704=1063.154,-79.560,437.949,171.659,25.481,154.745
C08705=1063.148,-79.810,437.960,171.657,25.479,154.745
C08706=1063.142,-80.059,437.971,171.656,25.478,154.745
C08707=1063.135,-80.309,437.982,171.654,25.476,154.745
C08708=1063.129,-80.558,437.993,171.652,25.475,154.745
C08709=1063.123,-80.808,438.005,171.651,25.473,154.745
C08710=1063.116,-81.057,438.015,171.649,25.472,154.745
C08711=1063.110,-81.307,438.026,171.647,25.470,154.745
C08712=1063.104,-81.557,438.037,171.646,25.469,154.745
C08713=1063.097,-81.807,438.048,171.644,25.467,154.745
C08714=1063.091,-82.089,438.060,171.642,25.466,154.745
C08715=1063.084,-82.370,438.072,171.640,25.464,154.744
C08716=1063.077,-82.652,438.084,171.638,25.462,154.744
C08717=1063.070,-82.934,438.097,171.637,25.461,154.744
C08718=1063.064,-83.184,438.108,171.635,25.459,154.744
C08719=1063.057,-83.434,438.118,171.633,25.458,154.744
C08720=1063.051,-83.683,438.129,171.631,25.456,154.744
C08721=1063.046,-83.933,438.140,171.629,25.454,154.744
C08722=1063.039,-84.183,438.151,171.627,25.453,154.744
C08723=1063.033,-84.432,438.162,171.626,25.452,154.744
C08724=1063.027,-84.682,438.173,171.624,25.450,154.744
C08725=1063.020,-84.931,438.183,171.622,25.449,154.744
C08726=1063.014,-85.181,438.194,171.621,25.448,154.744
C08727=1063.008,-85.431,438.205,171.619,25.446,154.744
C08728=1063.001,-85.680,438.216,171.617,25.445,154.744
C08729=1062.996,-85.930,438.226,171.615,25.443,154.744
C08730=1062.989,-86.180,438.238,171.614,25.442,154.744
C08731=1062.983,-86.430,438.247,171.612,25.440,154.744
C08732=1062.977,-86.679,438.258,171.610,25.439,154.744
C08733=1062.971,-86.930,438.269,171.609,25.437,154.743
C08734=1062.965,-87.179,438.280,171.607,25.436,154.743
C08735=1062.959,-87.428,438.291,171.605,25.435,154.743
C08736=1062.953,-87.678,438.302,171.604,25.433,154.743
C08737=1062.946,-87.928,438.312,171.602,25.432,154.743
C08738=1062.940,-88.177,438.323,171.600,25.431,154.743
C08739=1062.935,-88.427,438.333,171.599,25.429,154.743
C08740=1062.928,-88.677,438.344,171.596,25.428,154.743
C08741=1062.922,-88.927,438.355,171.594,25.426,154.743
C08742=1062.916,-89.176,438.366,171.593,25.425,154.743
C08743=1062.909,-89.426,438.376,171.591,25.423,154.743
C08744=1062.904,-89.676,438.386,171.589,25.422,154.743
C08745=1062.898,-89.925,438.397,171.588,25.421,154.743
C08746=1062.892,-90.175,438.407,171.586,25.420,154.743
C08747=1062.885,-90.425,438.419,171.584,25.418,154.743
C08748=1062.879,-90.674,438.429,171.583,25.417,154.743
C08749=1062.873,-90.924,438.439,171.581,25.416,154.743
C08750=1062.868,-91.174,438.450,171.579,25.414,154.743
C08751=1062.860,-91.423,438.461,171.578,25.413,154.742
C08752=1062.855,-91.673,438.472,171.576,25.411,154.742
C08753=1062.849,-91.923,438.482,171.574,25.410,154.742
C08754=1062.843,-92.172,438.492,171.572,25.409,154.742
C08755=1062.837,-92.422,438.503,171.571,25.407,154.742
C08756=1062.830,-92.672,438.513,171.569,25.406,154.742
C08757=1062.825,-92.922,438.524,171.567,25.405,154.742
C08758=1062.819,-93.171,438.535,171.566,25.404,154.742
C08759=1062.812,-93.420,438.545,171.564,25.402,154.742
C08760=1062.806,-93.671,438.555,171.562,25.400,154.742
C08761=1062.800,-93.920,438.566,171.560,25.399,154.742
C08762=1062.794,-94.170,438.577,171.558,25.398,154.742
C08763=1062.789,-94.420,438.587,171.556,25.397,154.742
C08764=1062.782,-94.669,438.597,171.555,25.395,154.742
C08765=1062.776,-94.919,438.608,171.553,25.394,154.742
C08766=1062.770,-95.169,438.618,171.551,25.392,154.742
C08767=1062.764,-95.419,438.629,171.550,25.391,154.742
C08768=1062.758,-95.668,438.638,171.548,25.390,154.742
C08769=1062.752,-95.918,438.649,171.546,25.389,154.742
C08770=1062.746,-96.167,438.660,171.544,25.388,154.742
C08771=1062.740,-96.418,438.670,171.543,25.386,154.742
C08772=1062.734,-96.667,438.681,171.541,25.385,154.742
C08773=1062.728,-96.917,438.690,171.539,25.384,154.742
C08774=1062.722,-97.167,438.701,171.538,25.382,154.742
C08775=1062.715,-97.416,438.712,171.536,25.381,154.742
C08776=1062.710,-97.666,438.722,171.534,25.380,154.742
C08777=1062.703,-97.916,438.732,171.533,25.379,154.742
C08778=1062.697,-98.200,438.744,171.530,25.377,154.742
C08779=1062.689,-98.484,438.755,171.528,25.376,154.742
C08780=1062.682,-98.768,438.767,171.526,25.375,154.742
C08781=1062.675,-99.052,438.779,171.524,25.373,154.742
C08782=1062.669,-99.302,438.789,171.522,25.372,154.742
C08783=1062.663,-99.552,438.800,171.520,25.371,154.742
C08784=1062.657,-99.802,438.809,171.519,25.369,154.742
C08785=1062.650,-100.051,438.820,171.517,25.368,154.742
C08786=1062.645,-100.301,438.830,171.515,25.367,154.742
C08787=1062.639,-100.551,438.839,171.513,25.366,154.742
C08788=1062.632,-100.800,438.850,171.512,25.365,154.742
C08789=1062.626,-101.051,438.860,171.510,25.364,154.742
C08790=1062.620,-101.300,438.870,171.508,25.363,154.742
C08791=1062.613,-101.550,438.880,171.507,25.362,154.742
C08792=1062.608,-101.799,438.891,171.505,25.360,154.742
C08793=1062.602,-102.049,438.900,171.503,25.359,154.742
C08794=1062.595,-102.298,438.911,171.501,25.358,154.742
C08795=1062.590,-102.548,438.921,171.500,25.357,154.741
C08796=1062.583,-102.798,438.930,171.498,25.356,154.742
C08797=1062.577,-103.047,438.941,171.496,25.355,154.742
C08798=1062.571,-103.298,438.951,171.494,25.354,154.742
C08799=1062.564,-103.547,438.961,171.493,25.352,154.742
C08800=1062.558,-103.797,438.971,171.491,25.351,154.742
C08801=1062.552,-104.047,438.981,171.488,25.350,154.742
C08802=1062.546,-104.296,438.991,171.486,25.349,154.742
C08803=1062.540,-104.546,439.001,171.485,25.348,154.742
C08804=1062.534,-104.796,439.011,171.483,25.347,154.742
C08805=1062.528,-105.045,439.021,171.481,25.345,154.742
C08806=1062.522,-105.295,439.031,171.480,25.344,154.742
C08807=1062.516,-105.545,439.041,171.478,25.344,154.742
C08808=1062.510,-105.794,439.051,171.476,25.342,154.742
C08809=1062.504,-106.044,439.061,171.474,25.341,154.742
C08810=1062.498,-106.294,439.071,171.473,25.340,154.742
C08811=1062.491,-106.543,439.081,171.471,25.339,154.742
C08812=1062.485,-106.794,439.091,171.469,25.338,154.742
C08813=1062.479,-107.044,439.101,171.467,25.337,154.742
C08814=1062.473,-107.294,439.111,171.466,25.336,154.742
C08815=1062.467,-107.543,439.121,171.464,25.335,154.742
C08816=1062.460,-107.793,439.130,171.462,25.334,154.742
C08817=1062.454,-108.042,439.140,171.460,25.333,154.742
C08818=1062.448,-108.292,439.150,171.458,25.332,154.742
C08819=1062.442,-108.541,439.160,171.457,25.331,154.742
C08820=1062.436,-108.791,439.170,171.455,25.330,154.742
C08821=1062.430,-109.041,439.180,171.453,25.329,154.742
C08822=1062.424,-109.291,439.189,171.451,25.328,154.742
C08823=1062.418,-109.541,439.199,171.450,25.327,154.742
C08824=1062.411,-109.790,439.209,171.448,25.326,154.742
C08825=1062.405,-110.040,439.219,171.445,25.324,154.742
C08826=1062.399,-110.290,439.228,171.443,25.324,154.742
C08827=1062.393,-110.539,439.238,171.442,25.323,154.742
C08828=1062.387,-110.790,439.248,171.440,25.322,154.742
C08829=1062.381,-111.039,439.258,171.438,25.321,154.742
C08830=1062.375,-111.289,439.268,171.436,25.320,154.742
C08831=1062.368,-111.538,439.277,171.434,25.319,154.742
C08832=1062.362,-111.788,439.287,171.433,25.318,154.742
C08833=1062.356,-112.038,439.296,171.431,25.317,154.742
C08834=1062.350,-112.288,439.306,171.429,25.316,154.742
C08835=1062.344,-112.538,439.316,171.427,25.315,154.743
C08836=1062.338,-112.787,439.325,171.426,25.314,154.742
C08837=1062.331,-113.036,439.335,171.424,25.313,154.743
C08838=1062.325,-113.286,439.345,171.422,25.312,154.743
C08839=1062.319,-113.536,439.355,171.420,25.312,154.743
C08840=1062.313,-113.786,439.365,171.418,25.310,154.743
C08841=1062.307,-114.036,439.374,171.417,25.310,154.743
C08842=1062.300,-114.318,439.385,171.415,25.309,154.743
C08843=1062.294,-114.601,439.396,171.412,25.307,154.743
C08844=1062.286,-114.883,439.406,171.410,25.306,154.743
C08845=1062.280,-115.165,439.418,171.409,25.305,154.743
C08846=1062.273,-115.415,439.427,171.407,25.305,154.743
C08847=1062.267,-115.664,439.436,171.405,25.304,154.743
C08848=1062.260,-115.914,439.446,171.403,25.303,154.743
C08849=1062.254,-116.164,439.455,171.401,25.302,154.743
C08850=1062.248,-116.414,439.465,171.400,25.301,154.743
C08851=1062.242,-116.664,439.474,171.397,25.300,154.743
C08852=1062.236,-116.913,439.484,171.395,25.299,154.743
C08853=1062.230,-117.163,439.494,171.393,25.298,154.743
C08854=1062.223,-117.413,439.503,171.392,25.297,154.744
C08855=1062.218,-117.662,439.512,171.390,25.296,154.743
C08856=1062.212,-117.912,439.522,171.388,25.296,154.744
C08857=1062.206,-118.162,439.531,171.386,25.295,154.744
C08858=1062.200,-118.412,439.540,171.384,25.294,154.744
C08859=1062.193,-118.662,439.550,171.383,25.293,154.744
C08860=1062.187,-118.912,439.559,171.381,25.293,154.744
C08861=1062.181,-119.161,439.569,171.379,25.291,154.744
C08862=1062.175,-119.411,439.579,171.377,25.291,154.744
C08863=1062.168,-119.661,439.588,171.375,25.290,154.744
C08864=1062.162,-119.911,439.597,171.373,25.289,154.744
C08865=1062.156,-120.160,439.606,171.372,25.288,154.744
C08866=1062.150,-120.409,439.616,171.370,25.288,154.744
C08867=1062.144,-120.659,439.625,171.368,25.287,154.744
C08868=1062.138,-120.910,439.634,171.366,25.286,154.744
C08869=1062.132,-121.159,439.644,171.364,25.285,154.744
C08870=1062.126,-121.409,439.653,171.363,25.285,154.745
C08871=1062.120,-121.659,439.663,171.361,25.284,154.745
C08872=1062.113,-121.908,439.672,171.359,25.283,154.745
C08873=1062.107,-122.158,439.681,171.357,25.282,154.745
C08874=1062.101,-122.408,439.690,171.355,25.281,154.745
C08875=1062.095,-122.658,439.700,171.353,25.281,154.745
C08876=1062.089,-122.908,439.709,171.352,25.280,154.745
C08877=1062.083,-123.157,439.719,171.350,25.279,154.745
C08878=1062.076,-123.406,439.727,171.348,25.278,154.745
C08879=1062.070,-123.657,439.736,171.346,25.278,154.745
C08880=1062.064,-123.906,439.746,171.344,25.277,154.745
C08881=1062.058,-124.156,439.755,171.342,25.276,154.746
C08882=1062.052,-124.406,439.765,171.341,25.276,154.746
C08883=1062.046,-124.656,439.774,171.339,25.275,154.746
C08884=1062.040,-124.905,439.782,171.337,25.274,154.746
C08885=1062.034,-125.155,439.792,171.335,25.273,154.746
C08886=1062.027,-125.405,439.802,171.333,25.273,154.746
C08887=1062.021,-125.655,439.810,171.331,25.272,154.746
C08888=1062.015,-125.905,439.819,171.330,25.272,154.746
C08889=1062.009,-126.154,439.829,171.327,25.271,154.746
C08890=1062.003,-126.404,439.838,171.325,25.270,154.746
C08891=1061.996,-126.654,439.846,171.323,25.269,154.746
C08892=1061.990,-126.904,439.856,171.321,25.269,154.747
C08893=1061.984,-127.153,439.865,171.319,25.268,154.747
C08894=1061.978,-127.403,439.873,171.318,25.267,154.747
C08895=1061.972,-127.653,439.883,171.316,25.267,154.747
C08896=1061.966,-127.902,439.893,171.314,25.266,154.747
C08897=1061.961,-128.152,439.902,171.312,25.264,154.747
C08898=1061.959,-128.403,439.912,171.311,25.263,154.747
C08899=1061.956,-128.654,439.924,171.310,25.261,154.746
C08900=1061.956,-128.905,439.936,171.309,25.258,154.746
C08901=1061.957,-129.155,439.949,171.308,25.254,154.746
C08902=1061.959,-129.407,439.962,171.307,25.249,154.745
C08903=1061.964,-129.658,439.976,171.306,25.244,154.744
C08904=1061.970,-129.909,439.991,171.306,25.239,154.743
C08905=1061.977,-130.159,440.007,171.306,25.233,154.742
C08906=1061.596,-130.181,439.818,171.258,25.388,154.775
C08907=1061.589,-129.932,439.803,171.258,25.394,154.776
C08908=1061.583,-129.681,439.787,171.259,25.400,154.777
C08909=1061.579,-129.430,439.773,171.259,25.404,154.778
C08910=1061.577,-129.178,439.759,171.260,25.409,154.779
C08911=1061.575,-128.927,439.747,171.261,25.413,154.779
C08912=1061.575,-128.677,439.734,171.262,25.416,154.779
C08913=1061.577,-128.425,439.723,171.264,25.418,154.780
C08914=1061.580,-128.175,439.713,171.265,25.420,154.780
C08915=1061.584,-127.925,439.702,171.267,25.421,154.780
C08916=1061.590,-127.675,439.693,171.269,25.422,154.780
C08917=1061.596,-127.426,439.685,171.271,25.423,154.780
C08918=1061.602,-127.176,439.675,171.273,25.423,154.780
C08919=1061.609,-126.926,439.666,171.274,25.424,154.780
C08920=1061.615,-126.676,439.657,171.276,25.425,154.779
C08921=1061.621,-126.426,439.648,171.278,25.425,154.779
C08922=1061.627,-126.177,439.639,171.280,25.426,154.779
C08923=1061.633,-125.927,439.629,171.282,25.426,154.779
C08924=1061.640,-125.677,439.621,171.284,25.428,154.779
C08925=1061.646,-125.428,439.611,171.285,25.428,154.779
C08926=1061.652,-125.178,439.602,171.287,25.429,154.779
C08927=1061.659,-124.928,439.593,171.289,25.429,154.779
C08928=1061.664,-124.679,439.584,171.291,25.430,154.779
C08929=1061.670,-124.429,439.575,171.293,25.431,154.779
C08930=1061.677,-124.179,439.565,171.295,25.431,154.779
C08931=1061.683,-123.929,439.556,171.297,25.432,154.778
C08932=1061.689,-123.679,439.547,171.298,25.433,154.778
C08933=1061.695,-123.430,439.538,171.300,25.434,154.778
C08934=1061.701,-123.180,439.529,171.302,25.434,154.778
C08935=1061.707,-122.930,439.519,171.304,25.435,154.778
C08936=1061.713,-122.680,439.510,171.306,25.436,154.778
C08937=1061.719,-122.430,439.501,171.308,25.436,154.778
C08938=1061.726,-122.181,439.492,171.309,25.437,154.778
C08939=1061.732,-121.932,439.482,171.311,25.438,154.778
C08940=1061.738,-121.682,439.473,171.313,25.439,154.778
C08941=1061.744,-121.432,439.463,171.315,25.439,154.778
C08942=1061.750,-121.182,439.454,171.317,25.441,154.778
C08943=1061.756,-120.932,439.445,171.318,25.441,154.778
C08944=1061.762,-120.682,439.435,171.320,25.442,154.777
C08945=1061.769,-120.432,439.426,171.322,25.442,154.777
C08946=1061.775,-120.183,439.417,171.325,25.444,154.777
C08947=1061.781,-119.934,439.407,171.327,25.444,154.777
C08948=1061.787,-119.684,439.398,171.329,25.445,154.777
C08949=1061.793,-119.434,439.388,171.330,25.446,154.777
C08950=1061.800,-119.184,439.379,171.332,25.447,154.777
C08951=1061.805,-118.934,439.370,171.334,25.448,154.777
C08952=1061.812,-118.684,439.360,171.336,25.448,154.777
C08953=1061.818,-118.434,439.351,171.338,25.449,154.777
C08954=1061.824,-118.184,439.341,171.339,25.450,154.777
C08955=1061.830,-117.935,439.332,171.341,25.451,154.777
C08956=1061.836,-117.686,439.322,171.343,25.452,154.777
C08957=1061.843,-117.436,439.313,171.345,25.452,154.777
C08958=1061.849,-117.186,439.304,171.347,25.453,154.776
C08959=1061.855,-116.936,439.294,171.348,25.454,154.776
C08960=1061.861,-116.687,439.285,171.350,25.455,154.776
C08961=1061.867,-116.437,439.275,171.352,25.456,154.776
C08962=1061.873,-116.187,439.266,171.354,25.457,154.776
C08963=1061.880,-115.937,439.256,171.356,25.457,154.776
C08964=1061.886,-115.687,439.247,171.357,25.459,154.776
C08965=1061.892,-115.438,439.237,171.359,25.459,154.776
C08966=1061.898,-115.188,439.227,171.361,25.460,154.776
C08967=1061.905,-114.906,439.216,171.364,25.461,154.776
C08968=1061.912,-114.623,439.206,171.365,25.462,154.776
C08969=1061.918,-114.341,439.195,171.367,25.463,154.776
C08970=1061.926,-114.058,439.184,171.369,25.464,154.776
C08971=1061.932,-113.809,439.174,171.371,25.465,154.776
C08972=1061.938,-113.559,439.165,171.374,25.466,154.776
C08973=1061.944,-113.309,439.155,171.375,25.467,154.776
C08974=1061.950,-113.059,439.145,171.377,25.468,154.776
C08975=1061.956,-112.809,439.136,171.379,25.469,154.775
C08976=1061.962,-112.560,439.126,171.381,25.470,154.776
C08977=1061.968,-112.310,439.116,171.383,25.471,154.775
C08978=1061.974,-112.060,439.107,171.384,25.472,154.775
C08979=1061.981,-111.811,439.097,171.386,25.472,154.775
C08980=1061.987,-111.561,439.087,171.388,25.474,154.775
C08981=1061.993,-111.311,439.077,171.390,25.475,154.775
C08982=1061.999,-111.061,439.068,171.391,25.476,154.775
C08983=1062.005,-110.812,439.058,171.393,25.477,154.775
C08984=1062.012,-110.562,439.049,171.395,25.477,154.775
C08985=1062.017,-110.312,439.039,171.397,25.479,154.775
C08986=1062.023,-110.063,439.028,171.399,25.479,154.775
C08987=1062.030,-109.813,439.019,171.400,25.480,154.775
C08988=1062.036,-109.563,439.009,171.402,25.482,154.775
C08989=1062.042,-109.313,439.000,171.404,25.482,154.775
C08990=1062.048,-109.063,438.990,171.406,25.483,154.775
C08991=1062.055,-108.814,438.980,171.407,25.485,154.775
C08992=1062.061,-108.564,438.970,171.409,25.485,154.775
C08993=1062.066,-108.314,438.960,171.411,25.486,154.775
C08994=1062.072,-108.065,438.950,171.413,25.487,154.775
C08995=1062.079,-107.815,438.940,171.415,25.489,154.775
C08996=1062.086,-107.565,438.930,171.417,25.490,154.775
C08997=1062.092,-107.315,438.921,171.419,25.490,154.775
C08998=1062.098,-107.065,438.911,171.421,25.492,154.775
C08999=1062.104,-106.816,438.900,171.422,25.493,154.775
C09000=1062.110,-106.566,438.891,171.424,25.494,154.775
C09001=1062.116,-106.316,438.881,171.426,25.495,154.775
C09002=1062.123,-106.067,438.871,171.428,25.496,154.775
C09003=1062.128,-105.817,438.861,171.430,25.497,154.775
C09004=1062.134,-105.567,438.851,171.431,25.498,154.775
C09005=1062.140,-105.317,438.842,171.433,25.499,154.775
C09006=1062.147,-105.068,438.831,171.435,25.500,154.775
C09007=1062.152,-104.818,438.821,171.437,25.501,154.775
C09008=1062.159,-104.569,438.811,171.438,25.502,154.775
C09009=1062.165,-104.319,438.801,171.440,25.504,154.775
C09010=1062.171,-104.069,438.792,171.442,25.504,154.775
C09011=1062.177,-103.820,438.781,171.444,25.505,154.775
C09012=1062.184,-103.569,438.771,171.445,25.507,154.775
C09013=1062.190,-103.319,438.761,171.447,25.508,154.775
C09014=1062.196,-103.070,438.750,171.449,25.509,154.775
C09015=1062.202,-102.820,438.741,171.451,25.510,154.775
C09016=1062.208,-102.571,438.731,171.452,25.511,154.775
C09017=1062.214,-102.321,438.720,171.455,25.512,154.775
C09018=1062.220,-102.071,438.711,171.457,25.514,154.775
C09019=1062.226,-101.822,438.701,171.458,25.515,154.775
C09020=1062.232,-101.572,438.690,171.460,25.516,154.775
C09021=1062.239,-101.322,438.680,171.462,25.517,154.775
C09022=1062.245,-101.072,438.670,171.464,25.518,154.775
C09023=1062.251,-100.823,438.659,171.465,25.519,154.775
C09024=1062.257,-100.573,438.650,171.467,25.520,154.775
C09025=1062.263,-100.324,438.639,171.469,25.521,154.775
C09026=1062.269,-100.074,438.629,171.471,25.523,154.775
C09027=1062.275,-99.824,438.619,171.472,25.524,154.775
C09028=1062.282,-99.574,438.609,171.474,25.525,154.775
C09029=1062.288,-99.324,438.598,171.476,25.526,154.775
C09030=1062.294,-99.075,438.589,171.477,25.527,154.775
C09031=1062.301,-98.790,438.577,171.480,25.529,154.775
C09032=1062.307,-98.506,438.566,171.482,25.530,154.775
C09033=1062.315,-98.222,438.554,171.484,25.531,154.775
C09034=1062.322,-97.938,438.542,171.486,25.533,154.775
C09035=1062.328,-97.688,438.532,171.488,25.534,154.775
C09036=1062.334,-97.439,438.521,171.490,25.535,154.775
C09037=1062.340,-97.189,438.512,171.491,25.536,154.775
C09038=1062.346,-96.939,438.500,171.493,25.538,154.775
C09039=1062.353,-96.689,438.491,171.495,25.539,154.775
C09040=1062.358,-96.439,438.480,171.496,25.541,154.775
C09041=1062.365,-96.190,438.470,171.498,25.542,154.775
C09042=1062.370,-95.940,438.460,171.500,25.543,154.775
C09043=1062.376,-95.691,438.449,171.502,25.544,154.775
C09044=1062.383,-95.441,438.438,171.503,25.545,154.775
C09045=1062.388,-95.191,438.428,171.505,25.547,154.775
C09046=1062.395,-94.941,438.418,171.507,25.548,154.775
C09047=1062.400,-94.691,438.407,171.509,25.549,154.775
C09048=1062.407,-94.442,438.397,171.510,25.551,154.775
C09049=1062.413,-94.193,438.386,171.512,25.552,154.775
C09050=1062.419,-93.942,438.376,171.514,25.553,154.775
C09051=1062.425,-93.693,438.365,171.515,25.554,154.775
C09052=1062.431,-93.443,438.355,171.517,25.556,154.775
C09053=1062.437,-93.194,438.344,171.519,25.557,154.775
C09054=1062.443,-92.944,438.334,171.521,25.559,154.775
C09055=1062.449,-92.694,438.323,171.523,25.560,154.775
C09056=1062.456,-92.445,438.313,171.525,25.561,154.775
C09057=1062.461,-92.194,438.302,171.526,25.562,154.775
C09058=1062.468,-91.945,438.292,171.528,25.564,154.775
C09059=1062.474,-91.695,438.281,171.530,25.565,154.776
C09060=1062.480,-91.446,438.270,171.531,25.567,154.776
C09061=1062.486,-91.196,438.261,171.533,25.568,154.776
C09062=1062.492,-90.946,438.250,171.535,25.569,154.776
C09063=1062.498,-90.696,438.238,171.537,25.571,154.776
C09064=1062.504,-90.447,438.228,171.538,25.572,154.776
C09065=1062.510,-90.197,438.218,171.540,25.573,154.776
C09066=1062.516,-89.948,438.208,171.542,25.574,154.776
C09067=1062.523,-89.697,438.196,171.543,25.576,154.776
C09068=1062.528,-89.448,438.186,171.545,25.577,154.776
C09069=1062.535,-89.199,438.175,171.547,25.579,154.776
C09070=1062.540,-88.949,438.165,171.548,25.580,154.776
C09071=1062.547,-88.698,438.154,171.550,25.582,154.776
C09072=1062.553,-88.449,438.144,171.552,25.583,154.776
C09073=1062.559,-88.200,438.133,171.554,25.584,154.776
C09074=1062.565,-87.950,438.121,171.556,25.586,154.776
C09075=1062.572,-87.700,438.111,171.558,25.587,154.776
C09076=1062.577,-87.451,438.100,171.560,25.588,154.776
C09077=1062.583,-87.200,438.090,171.561,25.590,154.776
C09078=1062.590,-86.951,438.079,171.563,25.591,154.776
C09079=1062.596,-86.701,438.069,171.565,25.593,154.776
C09080=1062.602,-86.451,438.057,171.566,25.594,154.776
C09081=1062.608,-86.202,438.047,171.568,25.596,154.777
C09082=1062.614,-85.953,438.036,171.570,25.597,154.777
C09083=1062.620,-85.702,438.025,171.571,25.598,154.777
C09084=1062.627,-85.453,438.015,171.573,25.600,154.777
C09085=1062.633,-85.204,438.004,171.575,25.601,154.777
C09086=1062.639,-84.954,437.993,171.576,25.603,154.777
C09087=1062.646,-84.704,437.982,171.578,25.604,154.777
C09088=1062.652,-84.454,437.972,171.580,25.605,154.777
C09089=1062.657,-84.204,437.961,171.581,25.607,154.777
C09090=1062.664,-83.955,437.951,171.583,25.608,154.777
C09091=1062.670,-83.705,437.939,171.585,25.609,154.777
C09092=1062.676,-83.455,437.928,171.587,25.611,154.777
C09093=1062.682,-83.206,437.918,171.589,25.613,154.777
C09094=1062.689,-82.956,437.907,171.591,25.614,154.777
C09095=1062.696,-82.674,437.895,171.592,25.616,154.777
C09096=1062.703,-82.392,437.882,171.594,25.617,154.778
C09097=1062.709,-82.110,437.870,171.597,25.619,154.778
C09098=1062.716,-81.829,437.857,171.598,25.621,154.778
C09099=1062.723,-81.579,437.846,171.600,25.622,154.778
C09100=1062.729,-81.329,437.836,171.602,25.624,154.778
C09101=1062.736,-81.079,437.824,171.603,25.625,154.778
C09102=1062.741,-80.830,437.813,171.605,25.627,154.778
C09103=1062.748,-80.580,437.803,171.607,25.628,154.778
C09104=1062.754,-80.330,437.792,171.608,25.630,154.778
C09105=1062.760,-80.081,437.781,171.610,25.631,154.778
C09106=1062.766,-79.831,437.770,171.612,25.632,154.778
